	5:	//MoveToTarget ready? -> Druck Ein
		fbMoveToTarget(bExecute:= TRUE);
		IF NOT fbMoveToTarget.bBusy THEN
			IF fbMoveToTarget.bError THEN
				stError.ErrorId := fbMoveToTarget.nErrorId;
				nActionState := 99;
			ELSE
				nActionState := 6;
			END_IF
			fbMoveToTarget(bExecute:= FALSE);
		END_IF	
		
	6:	//Switch Pressure
		IF pStampSupport^.M_GetPressValueOk(nSetPressure:= nPressure1, nTolerancePlus:= 8, nToleranceMinus:= 8) THEN 
			MEMSET(ADR(stActionData),0,SIZEOF(stActionData));
			stActionData.eAction := E_Action.ACTION_SwitchPressure;
			stActionData.aParams[1] := E_PressCtrl.PRESSCTRL_PressOn;
			stError.ErrorId := pStampSupport^.M_ExeAction(stActionData);
		ELSE
			stError.ErrorId := E_ErrorIdCmd.ERRORID_PressTimeOut;
		END_IF
		
		IF stError.ErrorId > 0 THEN	//Error
			stError.ObjectId := pStampSupport^.P_nObjectID;
			nActionState := 99;
		ELSE
			nActionState := 7;
		END_IF

	7:	//MoveZ um ContactDistance nach unten
		nActionState := 8;
		timer1(IN:=FALSE);
		MEMSET(ADR(stActionData),0,SIZEOF(stActionData));
		stActionData.eAction := E_Action.ACTION_MoveZ;
		stActionData.aParams[1] := E_MoveMode.MODE_Relative;
		stActionData.aParams[2] := - nDistance1;
		stActionData.aParams[3] := 1000;
		stError.ErrorId := pStampSupport^.M_ExeAction(stActionData);
		IF stError.ErrorId > 0 THEN	//Error
			stError.ObjectId := pStampSupport^.P_nObjectID;
			nActionState := 99;
		END_IF
		
	8:	//MoveZ ready? -> Timer starten
		IF NOT pStampSupport^.M_GetActionBusy(E_Action.ACTION_MoveZ) THEN
			timer1(IN:=TRUE, PT:= UDINT_TO_TIME(nTime));
			nActionState := 9;
		END_IF
		
	9:	//Warten, bis Zeit abgelaufen -> MoveZ um ContactDistance nach oben
		timer1();
		IF timer1.Q THEN
			nActionState := 10;
			MEMSET(ADR(stActionData),0,SIZEOF(stActionData));
			stActionData.eAction := E_Action.ACTION_MoveZ;
			stActionData.aParams[1] := E_MoveMode.MODE_Relative;
			stActionData.aParams[2] := nDistance1;
			stActionData.aParams[3] := 1000;			
			stError.ErrorId := pStampSupport^.M_ExeAction(stActionData);
			IF stError.ErrorId > 0 THEN	//Error
				stError.ObjectId := pStampSupport^.P_nObjectID;
				nActionState := 99;
			END_IF				
		END_IF
		
	10:	//MoveZ ready? -> Druck aus und MoveFree
		IF NOT pStampSupport^.M_GetActionBusy(E_Action.ACTION_MoveZ) THEN
			MEMSET(ADR(stActionData),0,SIZEOF(stActionData));
			stActionData.eAction := E_Action.ACTION_SwitchPressure;
			stActionData.aParams[1] := 1;
			stActionData.aParams[2] := E_PressCtrl.PRESSCTRL_Off;
			stError.ErrorId := pStampSupport^.M_ExeAction(stActionData);
			IF stError.ErrorId > 0 THEN	//Error
				stError.ObjectId := pStampSupport^.P_nObjectID;
				nActionState := 99;
			ELSE
				stActionData.eAction := E_Action.ACTION_MoveZ;
				stActionData.aParams[1] := E_MoveMode.MODE_Free;
				stActionData.aParams[3] := -1; //MaxSpeed Z
				stError.ErrorId := pStampSupport^.M_ExeAction(stActionData);
				IF stError.ErrorId > 0 THEN	//Error
					stError.ObjectId := pStampSupport^.P_nObjectID;
					nActionState := 99;
				ELSE
					nActionState := 11;
				END_IF			
			END_IF
		END_IF
		
	11:	//MoveZ-Free ready? -> Target = InkStation? -> CloseInkStation
		IF NOT pStampSupport^.M_GetActionBusy(E_Action.ACTION_MoveZ) THEN
			IF pInkStation > 0 THEN
				MEMSET(ADR(stActionData),0,SIZEOF(stActionData));
				stActionData.eAction := E_Action.ACTION_InkOpClCover;
				stActionData.aParams[1] := 1;
				stError.ErrorId := pInkStation^.M_ExeAction(stActionData);
				IF stError.ErrorId > 0 THEN
					stError.ObjectId := pTarget^.P_nObjectID;
					nActionState := 99;
				ELSE
					nActionState := 12;	
				END_IF
			ELSE
				nActionState := 80;
			END_IF
		END_IF
		
	12:	//Inkstation ready? -> Action ready
		IF NOT pInkStation^.M_GetActionBusy(E_Action.ACTION_InkOpClCover) THEN
			nActionState := 80;
		END_IF
		
	70:	//Abbrechen
		nActionState := 80;
		//MoveToTarget oder Einzel-Moves vom MzTool abbrechen (schließen sich gegenseitig aus)
		IF fbMoveToTarget.bBusy THEN
			fbMoveToTarget(bStop:= TRUE);
			nActionState := 70;
		ELSIF pStampSupport^.M_GetActionBusy(E_Action.ACTION_MoveZ) THEN
			pStampSupport^.M_CancelAction(E_Action.ACTION_MoveZ);
			nActionState := 70;
		ELSE
			fbMoveToTarget(bStop:= FALSE);
		END_IF
		
		IF pStampSupport^.M_GetActionBusy(E_Action.ACTION_SetPressure) THEN
			pStampSupport^.M_CancelAction(E_Action.ACTION_SetPressure);
			nActionState := 70;
		END_IF
		
		IF pStampSupport^.M_GetActionBusy(E_Action.ACTION_SwitchPressure) THEN
			pStampSupport^.M_CancelAction(E_Action.ACTION_SwitchPressure);
			nActionState := 70;
		END_IF
		
		//InkStation abbrechen
		IF pInkStation > 0 THEN
			IF pInkStation^.M_GetActionBusy(E_Action.ACTION_InkOpClCover) THEN
				pInkStation^.M_CancelAction(E_Action.ACTION_InkOpClCover);
				nActionState := 70;
			END_IF
		END_IF
END_CASE

//Errorhandling
IF nActionState = 99 THEN
	fbMoveToTarget(bExecute:= FALSE);
	stError.Cmd := E_Action.ACTION_StampInking;
	stError.POUAction := E_POUACT.POUACT_A_StampInking;
	fbErrorList.M_Add(stError);
END_IF
END_ACTION

ACTION A_TeachTarget:
stError.POUState := nActionState;

IF pMzTool^.P_bError THEN
	stError.ErrorId := pMzTool^.P_nErrorId;
	nActionState := 99;
END_IF

IF pMzTool^.P_bCanceled AND nActionState > 0 AND nActionState < 70 THEN
	//MzTool wurde durch StopDevice abgebrochen
	nActionState := 70;
END_IF

CASE nActionState OF
	0:	//MoveToTarget
		IF eTeachOption = E_TeachTrgtOption.Option_PrePos THEN
			MEMSET(ADR(stActionData),0,SIZEOF(stActionData));
			stActionData.eAction := E_Action.ACTION_MoveToTarget;
			stActionData.nObject := pMzTool^.P_nObjectID;
			stActionData.nTarget := pTarget^.P_nObjectID;
		
			IF pTarget^.P_eObjectType = E_ObjectType.OBJECTTYPE_Mtp THEN	//MoveToTarget Well1
				stActionData.aParams[1] := E_TargetRef.TARGETREF_TwoDimArray;
				stActionData.aParams[2] := 1; //Col (erstes Well immer Spalte 1)
				stActionData.aParams[3] := pMtp^.P_nRows; //Row (erstes Well immer letzte Spalte)
			ELSIF pTarget^.P_eObjectType = E_ObjectType.OBJECTTYPE_SpotArray THEN	//MoveToTarget Ecke links unten
				stActionData.aParams[1] := E_TargetRef.TARGETREF_LeftBottom;
			ELSIF pTarget^.P_eObjectType = E_ObjectType.OBJECTTYPE_Slide AND eTargetRef = E_TargetRef.TARGETREF_Alignment THEN	//MoveToTarget Alignment-Marke 1
				stActionData.aParams[1] := E_TargetRef.TARGETREF_SpecPoint;
				stActionData.aParams[2] := 1; //SpecPoint 1 (Marke 1)
			ELSE	//MoveToTarget Slot oder Center
				stActionData.aParams[1] := eTargetRef;
				stActionData.aParams[2] := nSpecPointSlotNr;
			END_IF
			stActionData.aParams[5] := -1;	//MaxSpeed X
			stActionData.aParams[6] := -1;	//MaxSpeed Y
			stActionData.aParams[7] := -1;	//MaxSpeed Z
			stActionData.aParams[10] := nZOffset1;
			stError.ErrorId := fbMoveToTarget.M_SetAndCheckParams(stActionData);
			IF stError.ErrorId > 0 THEN
				nActionState := 99;
			ELSE
				fbMoveToTarget(bExecute:= TRUE);
				nActionState := 1;
			END_IF
			
		ELSIF eTeachOption = E_TeachTrgtOption.Option_NoPrePos THEN
			//alle anderen Tools freifahren
			//dazu wird der Head benötigt:
			stError.ErrorId := pMzTool^.P_pMzHead^.M_MoveFree(pMzTool);
			IF stError.ErrorId > 0 THEN
				nActionState := 99;
			ELSE
				nActionState := 2;
			END_IF
			
		ELSIF eTeachOption = E_TeachTrgtOption.Option_AssumeInstantly THEN
			//aktuellen Wert sofort übernehmen
			stError.ErrorId := pTarget^.M_ApplyPos(eTargetRef, nSpecPointSlotNr, pMzTool^.P_stCurrentPosTotal, bXPos:= TRUE, bYPos:=TRUE, bZPos:=TRUE);
			IF stError.ErrorId > 0 THEN
				nActionState := 99;
			ELSE
				fbObjectDirectory.M_SetObjChange(pTarget^.P_nObjectID);
				nActionState := 80;
			END_IF
		ELSE
			{warnig 'ImplementErrorId'}
			stError.ErrorId := 333;
			nActionState := 99;
		END_IF
		MEMSET(ADR(stInteractRequest),0,SIZEOF(stInteractRequest));

	1:	//MoveToTarget ready?
		fbMoveToTarget(bExecute:= TRUE);
		IF NOT fbMoveToTarget.bBusy THEN
			IF fbMoveToTarget.bError THEN
				stError.ErrorId := fbMoveToTarget.nErrorId;
				nActionState := 99;
			ELSE
				nActionState := 2;	
			END_IF
			fbMoveToTarget(bExecute:= FALSE);
		END_IF
		
	2:	//Interaction Request "StartTeaching"
		IF NOT pMzTool^.P_pMzHead^.M_GetActionBusy(E_Action.ACTION_MoveZ) THEN
			MEMSET(ADR(stInterResponse),0,SIZEOF(stInterResponse));
			stInteractRequest.eInteractMessageType := E_InteractMessageType.INTERACTMES_StartTeaching;
			stInteractRequest.nObjectId := pMzTool^.P_nObjectID;
			stInteractRequest.nArg1 := 1;
			nActionState := 3;
		END_IF
		
	3:	//Response ?
		IF stInterResponse.eInteractMessageType = E_InteractMessageType.INTERACTMES_Assume THEN
			stInteractRequest.nArg1 := stInterResponse.nArg1;
			stInteractRequest.nArg2 := stInterResponse.nArg2;
			stInteractRequest.nArg3 := stInterResponse.nArg3; 
			
			pTarget^.M_ApplyPos(eTargetRef, nSpecPointSlotNr, pMzTool^.P_stCurrentPosTotal,
								bXPos:= DINT_TO_BOOL(stInterResponse.nArg1),
								bYPos:= DINT_TO_BOOL(stInterResponse.nArg2),
								bZPos:= DINT_TO_BOOL(stInterResponse.nArg3));

			fbObjectDirectory.M_SetObjChange(pTarget^.P_nObjectID);
			stInteractRequest.eInteractMessageType := E_InteractMessageType.INTERACTMES_Continue; //Request "Continue"
			MEMSET(ADR(stInterResponse),0,SIZEOF(stInterResponse));

		ELSIF stInterResponse.eInteractMessageType = E_InteractMessageType.INTERACTMES_TeachingFinished THEN
			IF pTarget^.P_eObjectType = E_ObjectType.OBJECTTYPE_Mtp AND eTargetRef = E_TargetRef.TARGETREF_TwoDimArray THEN
				pMtp^.M_CalcOffsetWellLB(pMzTool^.P_stCurrentPosTotal,0);
				stInteractRequest.eInteractMessageType := E_InteractMessageType.INTERACTMES_StartTeaching;	//Request "StartTeaching"
				stInteractRequest.nObjectId := pMzTool^.P_nObjectID;
				stInteractRequest.nArg1 := 2;
				nActionState := 4;
			ELSIF pTarget^.P_eObjectType = E_ObjectType.OBJECTTYPE_SpotArray AND eTargetRef = E_TargetRef.TARGETREF_TwoDimArray THEN
				//Position übertragen (nur XY)
				pTarget^.M_ApplyPos(eTargetRef:= E_TargetRef.TARGETREF_LeftBottom, 0, pMzTool^.P_stCurrentPosTotal,
									bXPos:= TRUE, bYPos:= TRUE, bZPos:= FALSE);
				IF eTeachOption = E_TeachTrgtOption.Option_NoPrePos THEN
					MEMSET(ADR(stInterResponse),0,SIZEOF(stInterResponse));
					stInteractRequest.eInteractMessageType := E_InteractMessageType.INTERACTMES_StartTeaching;	//Request "StartTeaching"
					stInteractRequest.nObjectId := pMzTool^.P_nObjectID;
					stInteractRequest.nArg1 := 2;
					nActionState := 9;
				ELSE
					nActionState := 7; //weiter zu MoveToTarget rechte obere Ecke
				END_IF
			(*
			ELSIF pTarget^.P_eObjectType = E_ObjectType.OBJECTTYPE_Slide AND eTargetRef = E_TargetRef.TARGETREF_Alignment THEN
				//Position auf Marke 1 übertragen
				pSlide := pTarget;
				pSlide^.M_SetMark1Act(pMzTool^.P_stCurrentPosTotal);
				nActionState := 10; //weiter zu MoveToTarget Alignment-Marke 2*)
			ELSE
				nActionState := 20; //weiter zu State "MoveZ-Free"
			END_IF
			MEMSET(ADR(stInterResponse),0,SIZEOF(stInterResponse));
		ELSIF stInterResponse.eInteractMessageType = E_InteractMessageType.INTERACTMES_Cancel THEN
			nActionState := 70;			
		END_IF
		
	//##################################################################################################################
	//Die nächsten 3 Schritte beziehen sich nur auf Mtp mit TargetRef "TwoDimArray"
	//##################################################################################################################
	4:	//Response "TeachingFinished"?
		IF stInterResponse.eInteractMessageType = E_InteractMessageType.INTERACTMES_TeachingFinished THEN
			MEMSET(ADR(stInteractRequest),0,SIZEOF(stInteractRequest));
			//Offset ermitteln und auf Well1 übertragen
			pMtp := pTarget;
			pMtp^.M_CalcOffsetWellLB(pMzTool^.P_stCurrentPosTotal,1);
			//MoveTo Target Wellx
			IF eTeachOption = E_TeachTrgtOption.Option_PrePos THEN
				MEMSET(ADR(stActionData),0,SIZEOF(stActionData));
				stActionData.eAction := E_Action.ACTION_MoveToTarget;
				stActionData.nObject := pMzTool^.P_nObjectID;
				stActionData.nTarget := pMtp^.P_nObjectID;
				stActionData.aParams[1] := E_TargetRef.TARGETREF_TwoDimArray;
				stActionData.aParams[2] := pMtp^.P_nCols; //Col (diagonales Well ermitteln)
				stActionData.aParams[3] := 1; //Row
				stActionData.aParams[5] := -1;	//MaxSpeed X
				stActionData.aParams[6] := -1;	//MaxSpeed Y
				stActionData.aParams[7] := -1;	//MaxSpeed Z
				stError.ErrorId := fbMoveToTarget.M_SetAndCheckParams(stActionData);
				IF stError.ErrorId > 0 THEN
					nActionState := 99;
				ELSE
					fbMoveToTarget(bExecute:= TRUE);
					nActionState := 5;
				END_IF
			ELSE
				MEMSET(ADR(stInterResponse),0,SIZEOF(stInterResponse));
				stInteractRequest.eInteractMessageType := E_InteractMessageType.INTERACTMES_StartTeaching;	//Request "StartTeaching"
				stInteractRequest.nObjectId := pMzTool^.P_nObjectID;
				stInteractRequest.nArg1 := 3;
				nActionState := 6;
			END_IF
		ELSIF stInterResponse.eInteractMessageType = E_InteractMessageType.INTERACTMES_Cancel THEN
			nActionState := 70;
		END_IF
		
	5:	//MoveToTarget ready?
		fbMoveToTarget(bExecute:= TRUE);
		IF NOT fbMoveToTarget.bBusy THEN
			IF fbMoveToTarget.bError THEN
				stError.ErrorId := fbMoveToTarget.nErrorId;
				nActionState := 99;
			ELSE
				MEMSET(ADR(stInterResponse),0,SIZEOF(stInterResponse));
				stInteractRequest.eInteractMessageType := E_InteractMessageType.INTERACTMES_StartTeaching;	//Request "StartTeaching"
				stInteractRequest.nObjectId := pMzTool^.P_nObjectID;
				stInteractRequest.nArg1 := 3;
				nActionState := 6;
			END_IF
			fbMoveToTarget(bExecute:= FALSE);
		END_IF	
		
	6:	//Response "TeachingFinished"?
		IF stInterResponse.eInteractMessageType = E_InteractMessageType.INTERACTMES_TeachingFinished THEN
			//Offset ermitteln und auf Wellx übertragen bzw. Korrekturfaktoren ermitteln
			pMtp^.M_CalcKorrFactor(pMzTool^.P_stCurrentPosTotal);
			nActionState := 20;
		ELSIF stInterResponse.eInteractMessageType = E_InteractMessageType.INTERACTMES_Cancel THEN
			nActionState := 70;
		END_IF
		//##################################################################################################################
		//Ende Teach Mtp Targetref "TwoDimArray
		//##################################################################################################################
		
		//##################################################################################################################
		//Die nächsten 3 Schritte beziehen sich nur auf SpotArray mit TargetRef "TwoDimArray"
		//##################################################################################################################
	7:	//MoveToTarget rechte obere Ecke
		MEMSET(ADR(stActionData),0,SIZEOF(stActionData));
		stActionData.eAction := E_Action.ACTION_MoveToTarget;
		stActionData.nObject := pMzTool^.P_nObjectID;
		stActionData.nTarget := pTarget^.P_nObjectID;
		stActionData.aParams[1] := E_TargetRef.TARGETREF_RightTop;
		stActionData.aParams[5] := -1;	//MaxSpeed X
		stActionData.aParams[6] := -1;	//MaxSpeed Y
		stActionData.aParams[7] := -1;	//MaxSpeed Z
		stActionData.aParams[10] := nZOffset1;
		stError.ErrorId := fbMoveToTarget.M_SetAndCheckParams(stActionData);
		IF stError.ErrorId > 0 THEN
			nActionState := 99;
		ELSE
			fbMoveToTarget(bExecute:= TRUE);
			nActionState := 8;
		END_IF
		
	8:	//MoveToTarget ready?
		fbMoveToTarget(bExecute:= TRUE);
		IF NOT fbMoveToTarget.bBusy THEN
			IF fbMoveToTarget.bError THEN
				stError.ErrorId := fbMoveToTarget.nErrorId;
				nActionState := 99;
			ELSE
				MEMSET(ADR(stInterResponse),0,SIZEOF(stInterResponse));
				stInteractRequest.eInteractMessageType := E_InteractMessageType.INTERACTMES_StartTeaching;	//Request "StartTeaching"
				stInteractRequest.nObjectId := pMzTool^.P_nObjectID;
				stInteractRequest.nArg1 := 2;
				nActionState := 9;
			END_IF
			fbMoveToTarget(bExecute:= FALSE);
		END_IF
		
	9:	//Response "TeachingFinished"?
		IF stInterResponse.eInteractMessageType = E_InteractMessageType.INTERACTMES_TeachingFinished THEN
			//Dimension in XY neu setzen
			stPoint1 := pTarget^.P_stAbsPosLB;
			stPoint2 := pMzTool^.P_stCurrentPosTotal;
			stDimension := pTarget^.P_stDimension;
			stDimension.Width := stPoint2.X - stPoint1.X;
			stDimension.Depth := stPoint2.Y - stPoint1.Y;
			pTarget^.P_stDimension := stDimension;
			nActionState := 20;
		ELSIF stInterResponse.eInteractMessageType = E_InteractMessageType.INTERACTMES_Cancel THEN
			nActionState := 70;
		END_IF	
		//##################################################################################################################
		//Ende Teach SpotArray Targetref "TwoDimArray
		//##################################################################################################################
		

		//##################################################################################################################
		//Die nächsten Schritte beziehen sich nur auf Slide mit TargetRef "Alignment"
		//##################################################################################################################
	10:	//MoveToTarget auf Alignment-Marke 2 Alignment gibt es nicht mehr
		(*
		MEMSET(ADR(stActionData),0,SIZEOF(stActionData));
		stActionData.eAction := E_Action.ACTION_MoveToTarget;
		stActionData.nObject := pMzTool^.P_nObjectID;
		stActionData.nTarget := pTarget^.P_nObjectID;
		stActionData.aParams[1] := E_TargetRef.TARGETREF_SpecPoint;
		stActionData.aParams[2] := 2;	//SpecPoint 1
		stActionData.aParams[5] := -1;	//MaxSpeed X
		stActionData.aParams[6] := -1;	//MaxSpeed Y
		stActionData.aParams[7] := -1;	//MaxSpeed Z
		stActionData.aParams[10] := nZOffset1;
		stError.ErrorId := fbMoveToTarget.M_SetAndCheckParams(stActionData);
		IF stError.ErrorId > 0 THEN
			nActionState := 99;
		ELSE
			fbMoveToTarget(bExecute:= TRUE);
			nActionState := 11;
		END_IF
	
	11:	//MoveToTarget ready?
		fbMoveToTarget(bExecute:= TRUE);
		IF NOT fbMoveToTarget.bBusy THEN
			IF fbMoveToTarget.bError THEN
				stError.ErrorId := fbMoveToTarget.nErrorId;
				nActionState := 99;
			ELSE
				MEMSET(ADR(stInterResponse),0,SIZEOF(stInterResponse));
				stInteractRequest.eInteractMessageType := E_InteractMessageType.INTERACTMES_StartTeaching;	//Request "StartTeaching"
				stInteractRequest.nObjectId := pMzTool^.P_nObjectID;
				stInteractRequest.nArg1 := 2;
				nActionState := 12;
			END_IF
			fbMoveToTarget(bExecute:= FALSE);
		END_IF 
	
	12:	//Response "TeachingFinished"?
		IF stInterResponse.eInteractMessageType = E_InteractMessageType.INTERACTMES_TeachingFinished THEN
			pSlide^.M_SetMark2Act(pMzTool^.P_stCurrentPosTotal);
			//Winkel berechnen
			pSlide^.P_bIsAligned := TRUE;
			pSlide^.M_CalcAngle();
			nActionState := 20;
		ELSIF stInterResponse.eInteractMessageType = E_InteractMessageType.INTERACTMES_Cancel THEN
			pSlide^.P_bIsAligned := FALSE;
			nActionState := 70;
		END_IF*)

	20:	//MoveZ-Free
		//Falls das Tool am unteren Head ist, dann freifahren überspringen.
		nActionState := 21;
		IF pMzTool^.P_pMzHead^.P_bIsTopHead THEN
			MEMSET(ADR(stActionData),0,SIZEOF(stActionData));
			stActionData.eAction := E_Action.ACTION_MoveZ;
			stActionData.aParams[1] := E_MoveMode.MODE_Free;
			stActionData.aParams[3] := -1;	//MaxSpeed Z
			stError.ErrorId := pMzTool^.M_ExeAction(stActionData);
			IF stError.ErrorId > 0 THEN
				nActionState := 99;
			END_IF
		END_IF
	
	21:	//MoveZ-Free ready? -> Action ready
		IF NOT pMzTool^.M_GetActionBusy(E_Action.ACTION_MoveZ) THEN
			fbObjectDirectory.M_SetObjChange(pTarget^.P_nObjectID);
			nActionState := 80;
			MEMSET(ADR(stInteractRequest),0,SIZEOF(stInteractRequest));
		END_IF
	
	70:	//Abbrechen
		IF fbMoveToTarget.bBusy THEN
			fbMoveToTarget(bStop:= TRUE);
		ELSIF pMzTool^.M_GetActionBusy(E_Action.ACTION_MoveZ) THEN
			pMzTool^.M_CancelAction(E_Action.ACTION_MoveZ);
		ELSE
			fbMoveToTarget(bExecute:= FALSE);
			MEMSET(ADR(stInteractRequest),0,SIZEOF(stInteractRequest));
			nActionState := 80;
		END_IF
END_CASE

//Errorhandling
IF nActionState = 99 THEN
	fbMoveToTarget(bExecute:= FALSE);
	stError.ObjectId := pMzTool^.P_nObjectID;
	stError.Cmd := E_Action.ACTION_TeachTarget;
	stError.POUAction := E_POUACT.POUACT_A_TeachTarget;
	fbErrorList.M_Add(stError);
END_IF
END_ACTION

ACTION A_TeachTool:
stError.POUState := nActionState;

IF pMzTool^.P_bError THEN
	stError.ErrorId := pMzTool^.P_nErrorId;
	nActionState := 99;
END_IF

IF pMzTool^.P_bCanceled AND nActionState > 0 AND nActionState < 70 THEN
	//MzTool wurde durch StopDevice abgebrochen
	nActionState := 70;
END_IF

CASE nActionState OF
	0:	//MoveToTarget
		MEMSET(ADR(stActionData),0,SIZEOF(stActionData));
		//stActionData.bIntern := TRUE;
		stActionData.eAction := E_Action.ACTION_MoveToTarget;
		stActionData.nObject := pMzTool^.P_nObjectID;
		stActionData.nTarget := pTarget^.P_nObjectID;
    	stActionData.aParams[1] := eTargetRef;
		stActionData.aParams[2] := nCol;
		stActionData.aParams[3] := nRow;
		stActionData.aParams[5] := -1;	//MaxSpeed X
		stActionData.aParams[6] := -1;	//MaxSpeed Y
		stActionData.aParams[7] := -1;	//MaxSpeed Z
		stActionData.aParams[10] := nZOffset1;		

		stError.ErrorId := fbMoveToTarget.M_SetAndCheckParams(stActionData);
		IF stError.ErrorId > 0 THEN
			nActionState := 99;
		ELSE
			fbMoveToTarget(bExecute:= TRUE);
			MEMSET(ADR(stInteractRequest),0,SIZEOF(stInteractRequest));
			nActionState := 1;
		END_IF		

	1:	//MoveToTarget ready? -> Request "StartTeaching"
		fbMoveToTarget(bExecute:= TRUE);
		IF NOT fbMoveToTarget.bBusy THEN
			IF fbMoveToTarget.bError THEN
				stError.ErrorId := fbMoveToTarget.nErrorId;
				nActionState := 99;
			ELSE
				MEMSET(ADR(stInterResponse),0,SIZEOF(stInterResponse));
				stInteractRequest.eInteractMessageType := E_InteractMessageType.INTERACTMES_StartTeaching;	//Interaction Request absenden
				stInteractRequest.nObjectId := pMzTool^.P_nObjectID;
				stInteractRequest.nArg1 := 1;
				nActionState := 2;
			END_IF
			fbMoveToTarget(bExecute:= FALSE);
		END_IF
	
	2:	//Zwischenschritt um stInteractRequest zurückzusetzen
		MEMSET(ADR(stInteractRequest),0,SIZEOF(stInteractRequest));
		nActionState := 3;

	3:	//Response ?
		IF stInterResponse.eInteractMessageType = E_InteractMessageType.INTERACTMES_Assume THEN
			//anhand von den Args von Response wird festgelegt, ob die Werte von X,Y,Z übernommen werden sollen
			//absolute Position (Sollposition)aus Target holen
			stPoint1 := pTarget^.M_GetAbsPos(pChildPos:= 0, eTargetRef:= eTargetRef,
												nParam1:= nCol, nParam2:= nRow, nParam3:= 0,nZLevel:= 0);			
			IF stInterResponse.nArg1 = 1 THEN
				pMzTool^.M_SetCurrentPos(1,stPoint1.X);
				stInteractRequest.nArg1 := 1;			
			END_IF

			IF stInterResponse.nArg2 = 1 THEN
				pMzTool^.M_SetCurrentPos(2,stPoint1.Y);
				stInteractRequest.nArg2 := 1;
			END_IF

			IF stInterResponse.nArg3 = 1 THEN
				pMzTool^.M_SetCurrentPos(3,stPoint1.Z);
				stInteractRequest.nArg3 := 1;
			END_IF
			stInteractRequest.eInteractMessageType := E_InteractMessageType.INTERACTMES_Continue;	//Request "Continue"
			MEMSET(ADR(stInterResponse),0,SIZEOF(stInterResponse));
		ELSIF stInterResponse.eInteractMessageType = E_InteractMessageType.INTERACTMES_TeachingFinished OR 
				stInterResponse.eInteractMessageType = E_InteractMessageType.INTERACTMES_Cancel THEN
			MEMSET(ADR(stInteractRequest),0,SIZEOF(stInteractRequest));
			MEMSET(ADR(stInterResponse),0,SIZEOF(stInterResponse));				
			nActionState := 80;
		END_IF

	70:	//Abbrechen
		IF fbMoveToTarget.bBusy THEN
			fbMoveToTarget(bStop:= TRUE);
		ELSE
			fbMoveToTarget(bExecute:= FALSE);
			MEMSET(ADR(stInteractRequest),0,SIZEOF(stInteractRequest));
			MEMSET(ADR(stInterResponse),0,SIZEOF(stInterResponse));
			nActionState := 80;
		END_IF		
END_CASE

//Errorhandling
IF nActionState = 99 THEN
	fbMoveToTarget(bExecute:= FALSE);
	stError.ObjectId := pMzTool^.P_nObjectID;
	stError.Cmd := E_Action.ACTION_TeachTool;
	stError.POUAction := E_POUACT.POUACT_A_TeachTool;
	fbErrorList.M_Add(stError);
END_IF
END_ACTION

ACTION A_TransferGas:
stError.POUState := nActionState;

IF pLuer^.P_bError THEN
	stError.ObjectId := pLuer^.P_nObjectID;
	stError.ErrorId := pLuer^.P_nErrorId;
	nActionState := 99;
ELSIF pLuer2^.P_bError THEN
	stError.ObjectId := pLuer2^.P_nObjectID;
	stError.ErrorId := pLuer2^.P_nErrorId;
	nActionState := 99;	
END_IF

IF (pLuer^.P_bCanceled OR pLuer2^.P_bCanceled) AND nActionState > 0 AND nActionState < 70 THEN
	//Ein MzTool wurde durch StopDevice abgebrochen
	nActionState := 70;
END_IF

CASE nActionState OF
	0:	//Voreinstellung Ventile

		//LuerSource
		//ValveDil on
		pLuer^.M_SwitchValveDiluter(TRUE);
		
		//ValveLuer off
		pLuer^.M_SwitchValveLuer(FALSE);
		
		//LuerDestination
		//ValveDil off
		pLuer2^.M_SwitchValveDiluter(FALSE);
		
		//ValveLuer on
		pLuer2^.M_SwitchValveLuer(TRUE);
		
		//Druck einstellen
		MEMSET(ADR(stActionData),0,SIZEOF(stActionData));
		stActionData.eAction := E_Action.ACTION_SetPressure;
		stActionData.aParams[1] := 1; //Fertigmeldung wenn Solldruck erreicht
		stActionData.aParams[2] := nPressure1; //Value in kPa
		stActionData.aParams[3] := 15; //Toleranz
		stActionData.aParams[4] := 15; //Toleranz
		stActionData.aParams[5] := 10000; //Timeout in ms
		stError.ErrorId :=  pLuer^.M_ExeAction(stActionData);
		IF stError.ErrorId > 0 THEN
			stError.ObjectId := pLuer^.P_nObjectID;
			nActionState := 99;
		ELSE
			nActionState := 1;
		END_IF
	
	1:	//Start Timer, ValveSynth.Gas "On"
		IF NOT pLuer^.M_GetActionBusy(E_Action.ACTION_SetPressure) THEN
			timer1(IN:=TRUE,PT:= DWORD_TO_TIME(nTime));
			pLuer^.M_SwitchValveSynthGas(TRUE);
			nActionState := 2;
		END_IF
		
	2:	//Timer ready? -> ValveSynth.Gas "Off"
		timer1();
		IF timer1.Q THEN
			timer1(IN:=FALSE);
			pLuer^.M_SwitchValveSynthGas(FALSE);
			pLuer^.M_SwitchValveDiluter(FALSE);
			pLuer2^.M_SwitchValveLuer(FALSE);
			nActionState := 80;
		END_IF
		
	70:	//Abbrechen
		nActionState := 80;
		IF pLuer^.M_GetActionBusy(E_Action.ACTION_SetPressure) THEN
			pLuer^.M_CancelAction(E_Action.ACTION_SetPressure);
			nActionState := 70;
		END_IF
		timer1(IN:=FALSE);
		pLuer^.M_SwitchValveSynthGas(FALSE);
		pLuer^.M_SwitchValveDiluter(FALSE);
		pLuer2^.M_SwitchValveLuer(FALSE);
END_CASE

//Errorhandling
IF nActionState = 99 THEN
	stError.Cmd := E_Action.ACTION_TransferGas;
	stError.POUAction := E_POUACT.POUACT_A_TransferGas;
	fbErrorList.M_Add(stError);
END_IF
END_ACTION

ACTION A_TransferLiquid:
stError.POUState := nActionState;

IF pDiluter1^.P_bError THEN
	stError.ErrorId := pDiluter1^.P_nErrorId;
	nActionState := 99;
END_IF

IF (pDiluter1^.P_bCanceled OR pLuer^.P_bCanceled OR pLuer2^.P_bCanceled) AND nActionState > 0 AND nActionState < 70 THEN
	//Ein MzTool wurde durch StopDevice abgebrochen
	nActionState := 70;
END_IF

CASE nActionState OF
	0:	//Voreinstellung Ventile
		//LuerSource
		//ValveDil on
		pLuer^.M_SwitchValveDiluter(TRUE);
		//ValveLuer on
		pLuer^.M_SwitchValveLuer(TRUE);
		//LuerDestination
		//ValveDil off
		pLuer2^.M_SwitchValveDiluter(TRUE);
		//ValveLuer on
		pLuer2^.M_SwitchValveLuer(TRUE);
		
		//Transfer am DilSource ausführen
		MEMSET(ADR(stActionData),0,SIZEOF(stActionData));
		stActionData.eAction := E_Action.ACTION_DilTransfer;
		stActionData.aParams[1] := pDiluter2^.P_nObjectID; //ObjectId DilDesti
		stActionData.aParams[2] := nQuantity1;
		stActionData.aParams[3] := nFlow1;
		stActionData.aParams[4] := nQuantity2;
		stActionData.aParams[5] := nQuantity3;

		stError.ErrorId :=  pDiluter1^.M_ExeAction(stActionData);
		IF stError.ErrorId > 0 THEN
			stError.ObjectId := pDiluter1^.P_nObjectID;
			nActionState := 99;
		ELSE
			nActionState := 1;
		END_IF		
		
	1:	//Transfer ready?
		IF NOT pDiluter1^.M_GetActionBusy(E_Action.ACTION_DilTransfer) THEN
			pLuer^.M_SwitchValveDiluter(FALSE);
			pLuer^.M_SwitchValveLuer(FALSE);
			pLuer2^.M_SwitchValveDiluter(FALSE);
			pLuer2^.M_SwitchValveLuer(FALSE);
			nActionState := 80;
		END_IF
	
	70:	//Abbrechen
		IF pDiluter1^.M_GetActionBusy(E_Action.ACTION_DilTransfer) THEN
			pDiluter1^.M_CancelAction(E_Action.ACTION_DilTransfer);
		ELSE
			pLuer^.M_SwitchValveDiluter(FALSE);
			pLuer^.M_SwitchValveLuer(FALSE);
			pLuer2^.M_SwitchValveDiluter(FALSE);
			pLuer2^.M_SwitchValveLuer(FALSE);
			nActionState := 80;			
		END_IF
END_CASE

//Errorhandling
IF nActionState = 99 THEN
	stError.Cmd := E_Action.ACTION_TransferLiquid;
	stError.POUAction := E_POUACT.POUACT_A_TransferLiquid;
	fbErrorList.M_Add(stError);
END_IF
END_ACTION

ACTION A_TransferTray:
//Mögliche Transfers
//-von linker Übergabestation zu TrayTransporterSlot
//-von rechter Übergabestation zu TrayTransporterSlot
//-von TrayTransporterSlot zu linker Übergabestation
//-von TrayTransporterSlot zu rechter Übergabestation

//Der Error muss für die States 0-2 hier gemeldet werden
//sonst erfolgt die Meldung aus den Sub-Actions
IF nActionState < 3 THEN
	IF pTrayTransporter^.P_bError THEN
		stError.ErrorId := pTrayTransporter^.P_nErrorId;
		stError.ObjectId := pTrayTransporter^.P_nObjectID;
		stError.Cmd := E_Action.ACTION_TransferTray;
		stError.POUAction := E_POUACT.POUACT_A_TransferTray;
		fbErrorList.M_Add(stError);
		nActionState := 99;	
	END_IF	
END_IF

IF nActionState > 0 AND nActionState < 70 AND pTrayTransporter^.P_bCanceled THEN
	nActionState := 70;
END_IF

CASE nActionState OF
	0:	//Both DrivingPins horizontal
		MEMSET(ADR(stActionData),0,SIZEOF(stActionData));
		stActionData.eAction := E_Action.ACTION_TurnDrivingPin;
		stActionData.nObject := pTrayTransporter^.P_nObjectID;
		stActionData.aParams[1] := E_DrivingPinSelection.Both;
		stActionData.aParams[2] := E_DrivingPinCtrl.Horizontal;
		stError.ErrorId := pTrayTransporter^.M_ExeAction(stActionData);
		IF stError.ErrorId > 0 THEN
			nActionState := 99;
		ELSE
			nActionState := 1;
		END_IF
		
	1:	//DrivingPins ready? -> Unlock TrayLock
		IF NOT pTrayTransporter^.M_GetActionBusy(E_Action.ACTION_TurnDrivingPin) THEN
			MEMSET(ADR(stActionData),0,SIZEOF(stActionData));
			stActionData.eAction := E_Action.ACTION_LockUnlock;
			stActionData.aParams[1] := E_LockCtrl.Unlock;
			stError.ErrorId := pTrayTransporter^.M_ExeAction(stActionData);
			IF stError.ErrorId > 0 THEN
				nActionState := 99;
			ELSE
				nActionState := 2;
			END_IF
		END_IF
		
	2:	//TrayLock ready?
		IF NOT pTrayTransporter^.M_GetActionBusy(E_Action.ACTION_LockUnlock) THEN
			IF pTrayTransporter^.P_bError THEN
				nActionState := 99;
			ELSE
				CASE eTransferTrayCtrl OF
					E_TransferTrayCtrl.LeftToSlot:
						nActionState := 3;
					E_TransferTrayCtrl.RightToSlot:
						nActionState := 4;
					E_TransferTrayCtrl.SlotToLeft:
						nActionState := 5;
					E_TransferTrayCtrl.SlotToRight:
						nActionState := 6;
				END_CASE
			END_IF
		END_IF
		
	3:	//Transfer left to slot
		A_TransferTrayLeftToSlot();
		IF nStateA_TransferTray >= 80 THEN
			IF nStateA_TransferTray = 99 THEN
				nActionState := 99;
			ELSE
				nActionState := 80;
			END_IF
			nStateA_TransferTray := 0;
		END_IF
	
	4:	//Transfer right to slot
		A_TransferTrayRightToSlot();
		IF nStateA_TransferTray >= 80 THEN
			IF nStateA_TransferTray = 99 THEN
				nActionState := 99;
			ELSE
				nActionState := 80;
			END_IF
			nStateA_TransferTray := 0;
		END_IF
	
	5:	//Transfer slot to left
		A_TransferTraySlotToLeft();
		IF nStateA_TransferTray >= 80 THEN
			IF nStateA_TransferTray = 99 THEN
				nActionState := 99;
			ELSE
				nActionState := 80;
			END_IF
			nStateA_TransferTray := 0;
		END_IF
	
	6:	//Transfer slot to right
		A_TransferTraySlotToRight();
		IF nStateA_TransferTray >= 80 THEN
			IF nStateA_TransferTray = 99 THEN
				nActionState := 99;
			ELSE
				nActionState := 80;
			END_IF
			nStateA_TransferTray := 0;
		END_IF
		
	70:	//Abbrechen
		IF pTrayTransporter^.P_bBusy THEN
			pTrayTransporter^.M_Stop();
		ELSE
			nStateA_TransferTray := 0;
			nActionState := 80;
		END_IF
END_CASE
END_ACTION

ACTION A_TransferTrayLeftToSlot:
CASE nStateA_TransferTray OF
	0:	//TransferStation ready for transfer?
		stError.ErrorId := pTrayTransporter^.M_GetStateForTransfer(E_TransferTrayCtrl.LeftToSlot);
		IF stError.ErrorId = 0 THEN
			nStateA_TransferTray := 1;
		ELSE
			nStateA_TransferTray := 99;
		END_IF
		
	1:	//Move slider TransferPosition left
		stActionData.eAction := E_Action.ACTION_MoveTrayTransporter;
		stActionData.aParams[1] := pTrayTransporter^.P_nTransferPosLeft;
		stActionData.aParams[2] := pTrayTransporter^.P_nMaxSliderSpeed;
		stError.ErrorId := pTrayTransporter^.M_ExeAction(stActionData);
		IF stError.ErrorId > 0 THEN
			nStateA_TransferTray := 99;
		ELSE
			nStateA_TransferTray := 2;
		END_IF
		
	2:	//Move ready? DrivingPin left vertical
		IF NOT pTrayTransporter^.M_GetActionBusy(E_Action.ACTION_MoveTrayTransporter) THEN
			stActionData.eAction := E_Action.ACTION_TurnDrivingPin;
			stActionData.aParams[1] := E_DrivingPinSelection.Left;
			stActionData.aParams[2] := E_DrivingPinCtrl.Vertical;
			stError.ErrorId := pTrayTransporter^.M_ExeAction(stActionData);
			IF stError.ErrorId > 0 THEN
				nStateA_TransferTray := 99;
			ELSE
				nStateA_TransferTray := 3;
			END_IF
		END_IF
		
	3:	//TurnDrivingPin ready? -> Move slider to slot + gap
		//Hier kann es sein, dass es nicht mit einem Zug geht.
		//Wenn also die TransferPos > als max SliderPos ist, dann wird zuerst bis max. Pos gefahren und dann über die mittlere Aussparung
		//das benötigt zusätzliche Steps
		IF NOT pTrayTransporter^.M_GetActionBusy(E_Action.ACTION_TurnDrivingPin) THEN
			stActionData.eAction := E_Action.ACTION_MoveTrayTransporter;
			nTransferTrayPos := pTrayTransporter^.M_GetSliderPosTrayInSlot(E_DrivingPinSelection.Left, E_TrayHollowSelection.Right) + pTrayTransporter^.P_nDrivingPinGap;
			IF nTransferTrayPos > pTrayTransporter^.P_nMaxSliderPos THEN
				nTransferTrayPos := pTrayTransporter^.P_nMaxSliderPos;
				nStateA_TransferTray := 4;
			ELSE
				nStateA_TransferTray := 20;
			END_IF
			stActionData.aParams[1] := nTransferTrayPos;
			stActionData.aParams[2] := cMoveTraySpeed;
			stError.ErrorId := pTrayTransporter^.M_ExeAction(stActionData);
			IF stError.ErrorId > 0 THEN
				nStateA_TransferTray := 99;
			END_IF
		END_IF
		
	4:	//Move ready? -> Move slider centre hollow (last pos - gap)
		IF NOT pTrayTransporter^.M_GetActionBusy(E_Action.ACTION_MoveTrayTransporter) THEN
			stActionData.eAction := E_Action.ACTION_MoveTrayTransporter;
			nTransferTrayPos :=  nTransferTrayPos - pTrayTransporter^.P_nDrivingPinGap;
			stActionData.aParams[1] := nTransferTrayPos;
			stActionData.aParams[2] := pTrayTransporter^.P_nMaxSliderSpeed;
			stError.ErrorId := pTrayTransporter^.M_ExeAction(stActionData);
			IF stError.ErrorId > 0 THEN
				nStateA_TransferTray := 99;
			ELSE
				nStateA_TransferTray := 5;
			END_IF
		END_IF
		
	5:	//Move ready? DrivingPinLeft horizontal
		IF NOT pTrayTransporter^.M_GetActionBusy(E_Action.ACTION_MoveTrayTransporter) THEN
			stActionData.eAction := E_Action.ACTION_TurnDrivingPin;
			stActionData.aParams[1] := E_DrivingPinSelection.Left;
			stActionData.aParams[2] := E_DrivingPinCtrl.Horizontal;
			stError.ErrorId := pTrayTransporter^.M_ExeAction(stActionData);
			IF stError.ErrorId > 0 THEN
				nStateA_TransferTray := 99;
			ELSE
				nStateA_TransferTray := 6;
			END_IF
		END_IF
		
	6:	//TurnDrivingPin ready? -> Move slider centre of tray (relative)
		IF NOT pTrayTransporter^.M_GetActionBusy(E_Action.ACTION_TurnDrivingPin) THEN
			stActionData.eAction := E_Action.ACTION_MoveTrayTransporter;
			nTransferTrayPos := nTransferTrayPos - pTrayTransporter^.P_nTrayLength /2 + pTrayTransporter^.P_nHollowDistance;
			stActionData.aParams[1] := nTransferTrayPos;
			stActionData.aParams[2] := pTrayTransporter^.P_nMaxSliderSpeed;
			stError.ErrorId := pTrayTransporter^.M_ExeAction(stActionData);
			IF stError.ErrorId > 0 THEN
				nStateA_TransferTray := 99;
			ELSE
				nStateA_TransferTray := 7;
			END_IF
		END_IF
		
	7:	//Move ready? DrivingPinLeft vertical
		IF NOT pTrayTransporter^.M_GetActionBusy(E_Action.ACTION_MoveTrayTransporter) THEN
			stActionData.eAction := E_Action.ACTION_TurnDrivingPin;
			stActionData.aParams[1] := E_DrivingPinSelection.Left;
			stActionData.aParams[2] := E_DrivingPinCtrl.Vertical;
			stError.ErrorId := pTrayTransporter^.M_ExeAction(stActionData);
			IF stError.ErrorId > 0 THEN
				nStateA_TransferTray := 99;
			ELSE
				nStateA_TransferTray := 8;
			END_IF
		END_IF
		
	8:	//TurnDrivingPin ready? -> Move slider to Slot
		IF NOT pTrayTransporter^.M_GetActionBusy(E_Action.ACTION_TurnDrivingPin) THEN
			stActionData.eAction := E_Action.ACTION_MoveTrayTransporter;
			nTransferTrayPos := pTrayTransporter^.M_GetSliderPosTrayInSlot(E_DrivingPinSelection.Left, E_TrayHollowSelection.Centre) + pTrayTransporter^.P_nDrivingPinGap;
			stActionData.aParams[1] := nTransferTrayPos;
			stActionData.aParams[2] := cMoveTraySpeed;
			stError.ErrorId := pTrayTransporter^.M_ExeAction(stActionData);
			IF stError.ErrorId > 0 THEN
				nStateA_TransferTray := 99;
			ELSE
				nStateA_TransferTray := 20;
			END_IF
		END_IF
		
	
	//Hier wird die Abzweigung in State "3" wieder zusammengeführt
		
	20:	//Move ready? -> Move slider centre hollow (last pos - gap)
		IF NOT pTrayTransporter^.M_GetActionBusy(E_Action.ACTION_MoveTrayTransporter) THEN
			stActionData.eAction := E_Action.ACTION_MoveTrayTransporter;
			stActionData.aParams[1] := nTransferTrayPos - pTrayTransporter^.P_nDrivingPinGap;
			stActionData.aParams[2] := pTrayTransporter^.P_nMaxSliderSpeed;
			stError.ErrorId := pTrayTransporter^.M_ExeAction(stActionData);
			IF stError.ErrorId > 0 THEN
				nStateA_TransferTray := 99;
			ELSE
				nStateA_TransferTray := 21;
			END_IF
		END_IF
		
	21:	//Move ready? DrivingPinLeft horizontal
		IF NOT pTrayTransporter^.M_GetActionBusy(E_Action.ACTION_MoveTrayTransporter) THEN
			stActionData.eAction := E_Action.ACTION_TurnDrivingPin;
			stActionData.aParams[1] := E_DrivingPinSelection.Left;
			stActionData.aParams[2] := E_DrivingPinCtrl.Horizontal;
			stError.ErrorId := pTrayTransporter^.M_ExeAction(stActionData);
			IF stError.ErrorId > 0 THEN
				nStateA_TransferTray := 99;
			ELSE
				nStateA_TransferTray := 22;
			END_IF
		END_IF

	22:	//TurnDrivingPin ready? -> Lock TrayLock
		IF NOT pTrayTransporter^.M_GetActionBusy(E_Action.ACTION_TurnDrivingPin) THEN
			stActionData.eAction := E_Action.ACTION_LockUnlock;
			stActionData.aParams[1] := E_LockCtrl.Lock;
			stError.ErrorId := pTrayTransporter^.M_ExeAction(stActionData);
			IF stError.ErrorId > 0 THEN
				nStateA_TransferTray := 99;
			ELSE
				nStateA_TransferTray := 23;
			END_IF
		END_IF
		
	23:	//TrayLock ready? -> Action ready
		IF NOT pTrayTransporter^.M_GetActionBusy(E_Action.ACTION_LockUnlock) THEN
			nStateA_TransferTray := 80;
		END_IF
END_CASE

//Errorhandling
IF nStateA_TransferTray = 99 THEN
	stError.Cmd := E_Action.ACTION_TransferTray;
	stError.POUAction := E_POUACT.POUACT_A_TransferTrayLeftToSlot;
	fbErrorList.M_Add(stError);	
END_IF
END_ACTION

ACTION A_TransferTrayRightToSlot:
CASE nStateA_TransferTray OF
	0:	//TransferStation ready for transfer?
		stError.ErrorId := pTrayTransporter^.M_GetStateForTransfer(E_TransferTrayCtrl.RightToSlot);
		IF stError.ErrorId = 0 THEN
			nStateA_TransferTray := 1;
		ELSE
			nStateA_TransferTray := 99;
		END_IF
		
	1:	//Move slider TransferPosition right
		stActionData.eAction := E_Action.ACTION_MoveTrayTransporter;
		stActionData.aParams[1] := pTrayTransporter^.P_nTransferPosRight;
		stActionData.aParams[2] := pTrayTransporter^.P_nMaxSliderSpeed;
		stError.ErrorId := pTrayTransporter^.M_ExeAction(stActionData);
		IF stError.ErrorId > 0 THEN
			nStateA_TransferTray := 99;
		ELSE
			nStateA_TransferTray := 2;
		END_IF
		
	2:	//Move ready? DrivingPin right vertical
		IF NOT pTrayTransporter^.M_GetActionBusy(E_Action.ACTION_MoveTrayTransporter) THEN
			stActionData.eAction := E_Action.ACTION_TurnDrivingPin;
			stActionData.aParams[1] := E_DrivingPinSelection.Right;
			stActionData.aParams[2] := E_DrivingPinCtrl.Vertical;
			stError.ErrorId := pTrayTransporter^.M_ExeAction(stActionData);
			IF stError.ErrorId > 0 THEN
				nStateA_TransferTray := 99;
			ELSE
				nStateA_TransferTray := 3;
			END_IF
		END_IF
		
	3:	//TurnDrivingPin ready? -> Move slider to SafePosLeft
		//Zuerst soweit wie möglich nach links fahren und dann um Abstand der äußeren Aussparungen wieder nach rechts fahren
		IF NOT pTrayTransporter^.M_GetActionBusy(E_Action.ACTION_TurnDrivingPin) THEN
			stActionData.eAction := E_Action.ACTION_MoveTrayTransporter;
			nTransferTrayPos := pTrayTransporter^.P_nSafePosLeft;
			stActionData.aParams[1] := nTransferTrayPos;
			stActionData.aParams[2] := cMoveTraySpeed;
			stError.ErrorId := pTrayTransporter^.M_ExeAction(stActionData);
			IF stError.ErrorId > 0 THEN
				nStateA_TransferTray := 99;
			ELSE
				nStateA_TransferTray := 4;
			END_IF
		END_IF
		
	4:	//Move ready? -> Move slider centre hollow (last pos + gap)
		IF NOT pTrayTransporter^.M_GetActionBusy(E_Action.ACTION_MoveTrayTransporter) THEN
			stActionData.eAction := E_Action.ACTION_MoveTrayTransporter;
			nTransferTrayPos :=  nTransferTrayPos + pTrayTransporter^.P_nDrivingPinGap;
			stActionData.aParams[1] := nTransferTrayPos;
			stActionData.aParams[2] := pTrayTransporter^.P_nMaxSliderSpeed;
			stError.ErrorId := pTrayTransporter^.M_ExeAction(stActionData);
			IF stError.ErrorId > 0 THEN
				nStateA_TransferTray := 99;
			ELSE
				nStateA_TransferTray := 5;
			END_IF
		END_IF
		
	5:	//Move ready? DrivingPinRight horizontal
		IF NOT pTrayTransporter^.M_GetActionBusy(E_Action.ACTION_MoveTrayTransporter) THEN
			stActionData.eAction := E_Action.ACTION_TurnDrivingPin;
			stActionData.aParams[1] := E_DrivingPinSelection.Right;
			stActionData.aParams[2] := E_DrivingPinCtrl.Horizontal;
			stError.ErrorId := pTrayTransporter^.M_ExeAction(stActionData);
			IF stError.ErrorId > 0 THEN
				nStateA_TransferTray := 99;
			ELSE
				nStateA_TransferTray := 6;
			END_IF
		END_IF
		
	6:	//Right hollow reachable?
		IF NOT pTrayTransporter^.M_GetActionBusy(E_Action.ACTION_TurnDrivingPin) THEN
			IF bAdditionalMoves THEN
				IF nTransferTrayPos + pTrayTransporter^.P_nHollowToHollow / 2 <= pTrayTransporter^.P_nMaxSliderPos THEN
					nStateA_TransferTray := 10;
				ELSE
					stError.ErrorId := E_ErrorIdCmd.ERRORID_CanNotTransferTrayCompletely;
					nStateA_TransferTray := 99; 
				END_IF
			ELSE
				IF nTransferTrayPos + pTrayTransporter^.P_nHollowToHollow <= pTrayTransporter^.P_nMaxSliderPos  THEN
					nStateA_TransferTray := 10;
				ELSE
					nStateA_TransferTray := 7;
				END_IF
			END_IF
		END_IF
		
	7:	//Move slider to middle hollow
		stActionData.eAction := E_Action.ACTION_MoveTrayTransporter;
		nTransferTrayPos := nTransferTrayPos + pTrayTransporter^.P_nTrayLength/2 - pTrayTransporter^.P_nHollowDistance;
		stActionData.aParams[1] := nTransferTrayPos;
		stActionData.aParams[2] := pTrayTransporter^.P_nMaxSliderSpeed;
		stError.ErrorId := pTrayTransporter^.M_ExeAction(stActionData);
		IF stError.ErrorId > 0 THEN
			nStateA_TransferTray := 99;
		ELSE
			nStateA_TransferTray := 8;
		END_IF
		
	8:	//Move ready? DrivingPin right vertical
		IF NOT pTrayTransporter^.M_GetActionBusy(E_Action.ACTION_MoveTrayTransporter) THEN
			stActionData.eAction := E_Action.ACTION_TurnDrivingPin;
			stActionData.aParams[1] := E_DrivingPinSelection.Right;
			stActionData.aParams[2] := E_DrivingPinCtrl.Vertical;
			stError.ErrorId := pTrayTransporter^.M_ExeAction(stActionData);
			IF stError.ErrorId > 0 THEN
				nStateA_TransferTray := 99;
			ELSE
				nStateA_TransferTray := 9;
			END_IF
		END_IF
		
	9:	//TurnDrivingPin ready? -> Move SafePosL
		IF NOT pTrayTransporter^.M_GetActionBusy(E_Action.ACTION_TurnDrivingPin) THEN
			stActionData.eAction := E_Action.ACTION_MoveTrayTransporter;
			nTransferTrayPos := pTrayTransporter^.P_nSafePosLeft;
			stActionData.aParams[1] := nTransferTrayPos;
			stActionData.aParams[2] := cMoveTraySpeed;
			stError.ErrorId := pTrayTransporter^.M_ExeAction(stActionData);
			IF stError.ErrorId > 0 THEN
				nStateA_TransferTray := 99;
			ELSE
				bAdditionalMoves := TRUE;
				nStateA_TransferTray := 4;
			END_IF
		END_IF

	10:	//TurnDrivingPin ready? -> Move slider at distance of both hollows (relative to previous position)
		stActionData.eAction := E_Action.ACTION_MoveTrayTransporter;
		IF bAdditionalMoves THEN //wird in State
			nTransferTrayPos := nTransferTrayPos + pTrayTransporter^.P_nHollowToHollow / 2;
		ELSE
			nTransferTrayPos := nTransferTrayPos + pTrayTransporter^.P_nHollowToHollow;	
		END_IF
		stActionData.aParams[1] := nTransferTrayPos;
		stActionData.aParams[2] := pTrayTransporter^.P_nMaxSliderSpeed;
		stError.ErrorId := pTrayTransporter^.M_ExeAction(stActionData);
		IF stError.ErrorId > 0 THEN
			nStateA_TransferTray := 99;
		ELSE
			nStateA_TransferTray := 11;
		END_IF
		
	11:	//Move ready? DrivingPinRight vertical
		IF NOT pTrayTransporter^.M_GetActionBusy(E_Action.ACTION_MoveTrayTransporter) THEN
			stActionData.eAction := E_Action.ACTION_TurnDrivingPin;
			stActionData.aParams[1] := E_DrivingPinSelection.Right;
			stActionData.aParams[2] := E_DrivingPinCtrl.Vertical;
			stError.ErrorId := pTrayTransporter^.M_ExeAction(stActionData);
			IF stError.ErrorId > 0 THEN
				nStateA_TransferTray := 99;
			ELSE
				nStateA_TransferTray := 12;
			END_IF
		END_IF
		
	12:	//TurnDrivingPin ready? -> Move slider to slot - DrivingPinGap
		IF NOT pTrayTransporter^.M_GetActionBusy(E_Action.ACTION_TurnDrivingPin) THEN
			stActionData.eAction := E_Action.ACTION_MoveTrayTransporter;
			nTransferTrayPos := pTrayTransporter^.M_GetSliderPosTrayInSlot(E_DrivingPinSelection.Right, E_TrayHollowSelection.Right) - pTrayTransporter^.P_nDrivingPinGap;
			stActionData.aParams[1] := nTransferTrayPos;
			stActionData.aParams[2] := cMoveTraySpeed;
			stError.ErrorId := pTrayTransporter^.M_ExeAction(stActionData);
			IF stError.ErrorId > 0 THEN
				nStateA_TransferTray := 99;
			ELSE
				nStateA_TransferTray := 13;
			END_IF
		END_IF
		
	13:	//Move ready? -> Move slider centre hollow (last pos - gap)
		IF NOT pTrayTransporter^.M_GetActionBusy(E_Action.ACTION_MoveTrayTransporter) THEN
			stActionData.eAction := E_Action.ACTION_MoveTrayTransporter;
			nTransferTrayPos :=  nTransferTrayPos + pTrayTransporter^.P_nDrivingPinGap;
			stActionData.aParams[1] := nTransferTrayPos;
			stActionData.aParams[2] := pTrayTransporter^.P_nMaxSliderSpeed;
			stError.ErrorId := pTrayTransporter^.M_ExeAction(stActionData);
			IF stError.ErrorId > 0 THEN
				nStateA_TransferTray := 99;
			ELSE
				nStateA_TransferTray := 14;
			END_IF
		END_IF

	14:	//Move ready? DrivingPinLeft horizontal
		IF NOT pTrayTransporter^.M_GetActionBusy(E_Action.ACTION_MoveTrayTransporter) THEN
			stActionData.eAction := E_Action.ACTION_TurnDrivingPin;
			stActionData.aParams[1] := E_DrivingPinSelection.Right;
			stActionData.aParams[2] := E_DrivingPinCtrl.Horizontal;
			stError.ErrorId := pTrayTransporter^.M_ExeAction(stActionData);
			IF stError.ErrorId > 0 THEN
				nStateA_TransferTray := 99;
			ELSE
				nStateA_TransferTray := 15;
			END_IF
		END_IF
		
	15:	//TurnDrivingPin ready? -> Lock TrayLock
		IF NOT pTrayTransporter^.M_GetActionBusy(E_Action.ACTION_TurnDrivingPin) THEN
			stActionData.eAction := E_Action.ACTION_LockUnlock;
			stActionData.aParams[1] := E_LockCtrl.Lock;
			stError.ErrorId := pTrayTransporter^.M_ExeAction(stActionData);
			IF stError.ErrorId > 0 THEN
				nStateA_TransferTray := 99;
			ELSE
				nStateA_TransferTray := 16;
			END_IF
		END_IF
		
	16:	//TrayLock ready? -> Action ready
		IF NOT pTrayTransporter^.M_GetActionBusy(E_Action.ACTION_LockUnlock) THEN
			nStateA_TransferTray := 80;
		END_IF		

END_CASE

//Errorhandling
IF nStateA_TransferTray = 99 THEN
	stError.Cmd := E_Action.ACTION_TransferTray;
	stError.POUAction := E_POUACT.POUACT_A_TransferTrayRightToSlot;
	fbErrorList.M_Add(stError);	
END_IF
END_ACTION

ACTION A_TransferTraySlotToLeft:
CASE nStateA_TransferTray OF
	0:	//TransferStation ready for transfer?
		stError.ErrorId := pTrayTransporter^.M_GetStateForTransfer(E_TransferTrayCtrl.SlotToLeft);
		IF stError.ErrorId = 0 THEN
			nStateA_TransferTray := 1;
		ELSE
			nStateA_TransferTray := 99;
		END_IF
		
	1:	//Move slider to slot
		//Hier kann es sein, dass zwei Züge erforderlich sind
		stActionData.eAction := E_Action.ACTION_MoveTrayTransporter;
		nTransferTrayPos := pTrayTransporter^.M_GetSliderPosTrayInSlot(E_DrivingPinSelection.Left, E_TrayHollowSelection.Right);
		IF nTransferTrayPos > pTrayTransporter^.P_nMaxSliderPos THEN //Mittlere Aussparung nutzen
			nTransferTrayPos := pTrayTransporter^.M_GetSliderPosTrayInSlot(E_DrivingPinSelection.Left, E_TrayHollowSelection.Centre);
			bAdditionalMoves := TRUE;
		ELSE
			bAdditionalMoves := FALSE;
		END_IF		
		stActionData.aParams[1] := nTransferTrayPos;
		stActionData.aParams[2] := pTrayTransporter^.P_nMaxSliderSpeed;
		stError.ErrorId := pTrayTransporter^.M_ExeAction(stActionData);
		IF stError.ErrorId > 0 THEN
			nStateA_TransferTray := 99;
		ELSE
			nStateA_TransferTray := 2;
		END_IF
		
	2:	//Move ready? DrivingPinLeft vertical
		IF NOT pTrayTransporter^.M_GetActionBusy(E_Action.ACTION_MoveTrayTransporter) THEN
			stActionData.eAction := E_Action.ACTION_TurnDrivingPin;
			stActionData.aParams[1] := E_DrivingPinSelection.Left;
			stActionData.aParams[2] := E_DrivingPinCtrl.Vertical;
			stError.ErrorId := pTrayTransporter^.M_ExeAction(stActionData);
			IF stError.ErrorId > 0 THEN
				nStateA_TransferTray := 99;
			ELSE
				nStateA_TransferTray := 3;
			END_IF
		END_IF
		
	3:	//TurnDrivingPin ready? -> Move slider TransferPosition left - DrivingPinGap
		IF NOT pTrayTransporter^.M_GetActionBusy(E_Action.ACTION_TurnDrivingPin) THEN
			stActionData.eAction := E_Action.ACTION_MoveTrayTransporter;
			nTransferTrayPos := pTrayTransporter^.P_nTransferPosLeft - pTrayTransporter^.P_nDrivingPinGap;
			stActionData.aParams[1] := nTransferTrayPos;
			stActionData.aParams[2] := cMoveTraySpeed;
			stError.ErrorId := pTrayTransporter^.M_ExeAction(stActionData);
			IF stError.ErrorId > 0 THEN
				nStateA_TransferTray := 99;
			ELSE
				nStateA_TransferTray := 4;
			END_IF
		END_IF
		
	4:	//Move ready? -> Move slider centre hollow (last pos + gap)
		IF NOT pTrayTransporter^.M_GetActionBusy(E_Action.ACTION_MoveTrayTransporter) THEN
			stActionData.eAction := E_Action.ACTION_MoveTrayTransporter;
			nTransferTrayPos := nTransferTrayPos + pTrayTransporter^.P_nDrivingPinGap;
			stActionData.aParams[1] := nTransferTrayPos;
			stActionData.aParams[2] := pTrayTransporter^.P_nMaxSliderSpeed;
			stError.ErrorId := pTrayTransporter^.M_ExeAction(stActionData);
			IF stError.ErrorId > 0 THEN
				nStateA_TransferTray := 99;
			ELSE
				nStateA_TransferTray := 5;
			END_IF
		END_IF
		
	5:	//Move ready? DrivingPinLeft horizontal
		IF NOT pTrayTransporter^.M_GetActionBusy(E_Action.ACTION_MoveTrayTransporter) THEN
			stActionData.eAction := E_Action.ACTION_TurnDrivingPin;
			stActionData.aParams[1] := E_DrivingPinSelection.Left;
			stActionData.aParams[2] := E_DrivingPinCtrl.Horizontal;
			stError.ErrorId := pTrayTransporter^.M_ExeAction(stActionData);
			IF stError.ErrorId > 0 THEN
				nStateA_TransferTray := 99;
			ELSE
				nStateA_TransferTray := 6;
			END_IF
		END_IF
		
	6:	//TurnDrivingPin ready? -> Move slider ??????
		//Slider muss jetzt um die Distanz von Mitte Ausssparung bis rechte Aussparung fahren
		//Achtung, Kommentar richtig stellen
		IF NOT pTrayTransporter^.M_GetActionBusy(E_Action.ACTION_TurnDrivingPin) THEN
			IF bAdditionalMoves THEN
				stActionData.eAction := E_Action.ACTION_MoveTrayTransporter;
				nTransferTrayPos := nTransferTrayPos + pTrayTransporter^.P_nTrayLength /2 - pTrayTransporter^.P_nHollowDistance;
				stActionData.aParams[1] := nTransferTrayPos;
				stActionData.aParams[2] := pTrayTransporter^.P_nMaxSliderSpeed;
				stError.ErrorId := pTrayTransporter^.M_ExeAction(stActionData);
				IF stError.ErrorId > 0 THEN
					nStateA_TransferTray := 99;
				ELSE
					nStateA_TransferTray := 7;
				END_IF
			ELSE
				nStateA_TransferTray := 11;
			END_IF
		END_IF
		
	7:	//Move ready? DrivingPinLeft vertical
		IF NOT pTrayTransporter^.M_GetActionBusy(E_Action.ACTION_MoveTrayTransporter) THEN
			stActionData.eAction := E_Action.ACTION_TurnDrivingPin;
			stActionData.aParams[1] := E_DrivingPinSelection.Left;
			stActionData.aParams[2] := E_DrivingPinCtrl.Vertical;
			stError.ErrorId := pTrayTransporter^.M_ExeAction(stActionData);
			IF stError.ErrorId > 0 THEN
				nStateA_TransferTray := 99;
			ELSE
				nStateA_TransferTray := 8;
			END_IF
		END_IF
		
	8:	//TurnDrivingPin ready? -> Move slider TransferPosLeft - DrivingPinGap
		IF NOT pTrayTransporter^.M_GetActionBusy(E_Action.ACTION_TurnDrivingPin) THEN
			stActionData.eAction := E_Action.ACTION_MoveTrayTransporter;
			nTransferTrayPos := pTrayTransporter^.P_nTransferPosLeft - pTrayTransporter^.P_nDrivingPinGap;
			stActionData.aParams[1] := nTransferTrayPos;
			stActionData.aParams[2] := pTrayTransporter^.P_nMaxSliderSpeed;
			stError.ErrorId := pTrayTransporter^.M_ExeAction(stActionData);
			IF stError.ErrorId > 0 THEN
				nStateA_TransferTray := 99;
			ELSE
				nStateA_TransferTray := 9;
			END_IF
		END_IF
		
	9:	//Move ready? -> Move slider centre hollow (last pos + gap)
		IF NOT pTrayTransporter^.M_GetActionBusy(E_Action.ACTION_MoveTrayTransporter) THEN
			stActionData.eAction := E_Action.ACTION_MoveTrayTransporter;
			nTransferTrayPos := nTransferTrayPos + pTrayTransporter^.P_nDrivingPinGap;
			stActionData.aParams[1] := nTransferTrayPos;
			stActionData.aParams[2] := pTrayTransporter^.P_nMaxSliderSpeed;
			stError.ErrorId := pTrayTransporter^.M_ExeAction(stActionData);
			IF stError.ErrorId > 0 THEN
				nStateA_TransferTray := 99;
			ELSE
				nStateA_TransferTray := 10;
			END_IF
		END_IF		
		
	10:	//Move ready? DrivingPinLeft horizontal
		IF NOT pTrayTransporter^.M_GetActionBusy(E_Action.ACTION_MoveTrayTransporter) THEN
			stActionData.eAction := E_Action.ACTION_TurnDrivingPin;
			stActionData.aParams[1] := E_DrivingPinSelection.Left;
			stActionData.aParams[2] := E_DrivingPinCtrl.Horizontal;
			stError.ErrorId := pTrayTransporter^.M_ExeAction(stActionData);
			IF stError.ErrorId > 0 THEN
				nStateA_TransferTray := 99;
			ELSE
				nStateA_TransferTray := 11;
			END_IF
		END_IF
		
	11:	//TurnDrivingPin ready? -> Move slider SafePosLeft
		IF NOT pTrayTransporter^.M_GetActionBusy(E_Action.ACTION_TurnDrivingPin) THEN
			stActionData.eAction := E_Action.ACTION_MoveTrayTransporter;
			nTransferTrayPos := pTrayTransporter^.P_nSafePosLeft;
			stActionData.aParams[1] := nTransferTrayPos;
			stActionData.aParams[2] := pTrayTransporter^.P_nMaxSliderSpeed;
			stError.ErrorId := pTrayTransporter^.M_ExeAction(stActionData);
			IF stError.ErrorId > 0 THEN
				nStateA_TransferTray := 99;
			ELSE
				nStateA_TransferTray := 12;
			END_IF
		END_IF
		
	12:	//TurnDrivingPin ready? -> Action ready
		IF NOT pTrayTransporter^.M_GetActionBusy(E_Action.ACTION_MoveTrayTransporter) THEN
			nStateA_TransferTray := 80;
		END_IF		
	
END_CASE

//Errorhandling
IF nStateA_TransferTray = 99 THEN
	stError.Cmd := E_Action.ACTION_TransferTray;
	stError.POUAction := E_POUACT.POUACT_A_TransferTraySlotToLeft;
	fbErrorList.M_Add(stError);	
END_IF
END_ACTION

ACTION A_TransferTraySlotToRight:
CASE nStateA_TransferTray OF
	0:	//TransferStation ready for transfer?
		stError.ErrorId := pTrayTransporter^.M_GetStateForTransfer(E_TransferTrayCtrl.SlotToRight);
		IF stError.ErrorId = 0 THEN
			nStateA_TransferTray := 1;
		ELSE
			nStateA_TransferTray := 99;
		END_IF
		
	1:	//Move slider to slot (right hollow with right driving pin)
		stActionData.eAction := E_Action.ACTION_MoveTrayTransporter;
		stActionData.aParams[1] := pTrayTransporter^.M_GetSliderPosTrayInSlot(E_DrivingPinSelection.Right, E_TrayHollowSelection.Right);
		stActionData.aParams[2] := pTrayTransporter^.P_nMaxSliderSpeed;
		stError.ErrorId := pTrayTransporter^.M_ExeAction(stActionData);
		IF stError.ErrorId > 0 THEN
			nStateA_TransferTray := 99;
		ELSE
			nStateA_TransferTray := 2;
		END_IF
		
	2:	//Move ready? DrivingPinLeft vertical
		IF NOT pTrayTransporter^.M_GetActionBusy(E_Action.ACTION_MoveTrayTransporter) THEN
			stActionData.eAction := E_Action.ACTION_TurnDrivingPin;
			stActionData.aParams[1] := E_DrivingPinSelection.Right;
			stActionData.aParams[2] := E_DrivingPinCtrl.Vertical;
			stError.ErrorId := pTrayTransporter^.M_ExeAction(stActionData);
			IF stError.ErrorId > 0 THEN
				nStateA_TransferTray := 99;
			ELSE
				nStateA_TransferTray := 3;
			END_IF
		END_IF
		
	3:	//Move slider TransferPosition right
		IF NOT pTrayTransporter^.M_GetActionBusy(E_Action.ACTION_TurnDrivingPin) THEN
			stActionData.eAction := E_Action.ACTION_MoveTrayTransporter;
			nTransferTrayPos := pTrayTransporter^.P_nTransferPosRight;
			stActionData.aParams[1] := nTransferTrayPos;
			stActionData.aParams[2] := cMoveTraySpeed;
			stError.ErrorId := pTrayTransporter^.M_ExeAction(stActionData);
			IF stError.ErrorId > 0 THEN
				nStateA_TransferTray := 99;
			ELSE
				nStateA_TransferTray := 4;
			END_IF		
		END_IF
		
	4:	//Move ready? -> Move slider centre hollow (last pos + gap)
		IF NOT pTrayTransporter^.M_GetActionBusy(E_Action.ACTION_MoveTrayTransporter) THEN
			stActionData.eAction := E_Action.ACTION_MoveTrayTransporter;
			nTransferTrayPos :=  nTransferTrayPos - pTrayTransporter^.P_nDrivingPinGap;
			stActionData.aParams[1] := nTransferTrayPos;
			stActionData.aParams[2] := pTrayTransporter^.P_nMaxSliderSpeed;
			stError.ErrorId := pTrayTransporter^.M_ExeAction(stActionData);
			IF stError.ErrorId > 0 THEN
				nStateA_TransferTray := 99;
			ELSE
				nStateA_TransferTray := 5;
			END_IF
		END_IF
		
	5:	//Move ready? DrivingPinRight horizontal
		IF NOT pTrayTransporter^.M_GetActionBusy(E_Action.ACTION_MoveTrayTransporter) THEN
			stActionData.eAction := E_Action.ACTION_TurnDrivingPin;
			stActionData.aParams[1] := E_DrivingPinSelection.Right;
			stActionData.aParams[2] := E_DrivingPinCtrl.Horizontal;
			stError.ErrorId := pTrayTransporter^.M_ExeAction(stActionData);
			IF stError.ErrorId > 0 THEN
				nStateA_TransferTray := 99;
			ELSE
				nStateA_TransferTray := 6;
			END_IF
		END_IF
		
	6:	//Left hollow reachable?
		IF NOT pTrayTransporter^.M_GetActionBusy(E_Action.ACTION_TurnDrivingPin) THEN
			IF bAdditionalMoves THEN
				IF nTransferTrayPos - pTrayTransporter^.P_nHollowToHollow / 2 >= pTrayTransporter^.P_nMinSliderPos THEN
					nStateA_TransferTray := 10;
				ELSE
					stError.ErrorId := E_ErrorIdCmd.ERRORID_CanNotTransferTrayCompletely;
					nStateA_TransferTray := 99; 
				END_IF
			ELSE
				IF nTransferTrayPos - pTrayTransporter^.P_nHollowToHollow >= pTrayTransporter^.P_nMinSliderPos  THEN
					nStateA_TransferTray := 10;
				ELSE
					nStateA_TransferTray := 7;
				END_IF
			END_IF
		END_IF
		
	7:	//Move slider to middle hollow
		stActionData.eAction := E_Action.ACTION_MoveTrayTransporter;
		nTransferTrayPos := nTransferTrayPos - pTrayTransporter^.P_nTrayLength/2 + pTrayTransporter^.P_nHollowDistance;
		stActionData.aParams[1] := nTransferTrayPos;
		stActionData.aParams[2] := pTrayTransporter^.P_nMaxSliderSpeed;
		stError.ErrorId := pTrayTransporter^.M_ExeAction(stActionData);
		IF stError.ErrorId > 0 THEN
			nStateA_TransferTray := 99;
		ELSE
			nStateA_TransferTray := 8;
		END_IF
		
	8:	//Move ready? DrivingPin right vertical
		IF NOT pTrayTransporter^.M_GetActionBusy(E_Action.ACTION_MoveTrayTransporter) THEN
			stActionData.eAction := E_Action.ACTION_TurnDrivingPin;
			stActionData.aParams[1] := E_DrivingPinSelection.Right;
			stActionData.aParams[2] := E_DrivingPinCtrl.Vertical;
			stError.ErrorId := pTrayTransporter^.M_ExeAction(stActionData);
			IF stError.ErrorId > 0 THEN
				nStateA_TransferTray := 99;
			ELSE
				nStateA_TransferTray := 9;
			END_IF
		END_IF
		
	9:	//TurnDrivingPin ready? -> Move TransferPosR
		IF NOT pTrayTransporter^.M_GetActionBusy(E_Action.ACTION_TurnDrivingPin) THEN
			stActionData.eAction := E_Action.ACTION_MoveTrayTransporter;
			nTransferTrayPos := pTrayTransporter^.P_nTransferPosRight;
			stActionData.aParams[1] := nTransferTrayPos;
			stActionData.aParams[2] := cMoveTraySpeed;
			stError.ErrorId := pTrayTransporter^.M_ExeAction(stActionData);
			IF stError.ErrorId > 0 THEN
				nStateA_TransferTray := 99;
			ELSE
				bAdditionalMoves := TRUE;
				nStateA_TransferTray := 4;
			END_IF
		END_IF
		
	10:	//TurnDrivingPin ready? -> Move slider at distance of both hollows (relative to previous position)
		stActionData.eAction := E_Action.ACTION_MoveTrayTransporter;
		IF bAdditionalMoves THEN //wird in State
			nTransferTrayPos := nTransferTrayPos - pTrayTransporter^.P_nHollowToHollow / 2;
		ELSE
			nTransferTrayPos := nTransferTrayPos - pTrayTransporter^.P_nHollowToHollow;	
		END_IF
		stActionData.aParams[1] := nTransferTrayPos;
		stActionData.aParams[2] := pTrayTransporter^.P_nMaxSliderSpeed;
		stError.ErrorId := pTrayTransporter^.M_ExeAction(stActionData);
		IF stError.ErrorId > 0 THEN
			nStateA_TransferTray := 99;
		ELSE
			nStateA_TransferTray := 11;
		END_IF
		
	11:	//Move ready? DrivingPinRight vertical
		IF NOT pTrayTransporter^.M_GetActionBusy(E_Action.ACTION_MoveTrayTransporter) THEN
			stActionData.eAction := E_Action.ACTION_TurnDrivingPin;
			stActionData.aParams[1] := E_DrivingPinSelection.Right;
			stActionData.aParams[2] := E_DrivingPinCtrl.Vertical;
			stError.ErrorId := pTrayTransporter^.M_ExeAction(stActionData);
			IF stError.ErrorId > 0 THEN
				nStateA_TransferTray := 99;
			ELSE
				nStateA_TransferTray := 12;
			END_IF
		END_IF
		
	12:	//TurnDrivingPin ready? -> Move TransferPosR + DrivingPinGap
		IF NOT pTrayTransporter^.M_GetActionBusy(E_Action.ACTION_TurnDrivingPin) THEN
			stActionData.eAction := E_Action.ACTION_MoveTrayTransporter;
			nTransferTrayPos := pTrayTransporter^.P_nTransferPosRight + pTrayTransporter^.P_nDrivingPinGap;
			stActionData.aParams[1] := nTransferTrayPos;
			stActionData.aParams[2] := cMoveTraySpeed;
			stError.ErrorId := pTrayTransporter^.M_ExeAction(stActionData);
			IF stError.ErrorId > 0 THEN
				nStateA_TransferTray := 99;
			ELSE
				nStateA_TransferTray := 13;
			END_IF
		END_IF
		
	13:	//Move ready? -> Move slider centre hollow (last pos + gap)
		IF NOT pTrayTransporter^.M_GetActionBusy(E_Action.ACTION_MoveTrayTransporter) THEN
			stActionData.eAction := E_Action.ACTION_MoveTrayTransporter;
			nTransferTrayPos :=  nTransferTrayPos - pTrayTransporter^.P_nDrivingPinGap;
			stActionData.aParams[1] := nTransferTrayPos;
			stActionData.aParams[2] := pTrayTransporter^.P_nMaxSliderSpeed;
			stError.ErrorId := pTrayTransporter^.M_ExeAction(stActionData);
			IF stError.ErrorId > 0 THEN
				nStateA_TransferTray := 99;
			ELSE
				nStateA_TransferTray := 14;
			END_IF
		END_IF
		
	14:	//Move ready? DrivingPinRight horizontal
		IF NOT pTrayTransporter^.M_GetActionBusy(E_Action.ACTION_MoveTrayTransporter) THEN
			stActionData.eAction := E_Action.ACTION_TurnDrivingPin;
			stActionData.aParams[1] := E_DrivingPinSelection.Right;
			stActionData.aParams[2] := E_DrivingPinCtrl.Horizontal;
			stError.ErrorId := pTrayTransporter^.M_ExeAction(stActionData);
			IF stError.ErrorId > 0 THEN
				nStateA_TransferTray := 99;
			ELSE
				nStateA_TransferTray := 15;
			END_IF
		END_IF
		
	15:	//TurnDrivingPin ready? -> Action ready
		IF NOT pTrayTransporter^.M_GetActionBusy(E_Action.ACTION_TurnDrivingPin) THEN
			nStateA_TransferTray := 80;
		END_IF		
		
END_CASE

//Errorhandling
IF nStateA_TransferTray = 99 THEN
	stError.Cmd := E_Action.ACTION_TransferTray;
	stError.POUAction := E_POUACT.POUACT_A_TransferTraySlotToRight;
	fbErrorList.M_Add(stError);	
END_IF
END_ACTION

ACTION A_WashTool:
stError.POUState := nActionState;

IF pMzTool^.P_bError THEN
	stError.ObjectId := pMzTool^.P_nObjectID;
	stError.ErrorId := pMzTool^.P_nErrorId;
	nActionState := 99;	
ELSIF pWashStation^.P_bError THEN
	stError.ObjectId := pWashStation^.P_nObjectID;
	stError.ErrorId := pWashStation^.P_nErrorId;
	nActionState := 99;
END_IF

CASE nActionState OF
	0:	//MoveToTarget "Washpoint"
		MEMSET(ADR(stActionData),0,SIZEOF(stActionData));
		stActionData.eAction := E_Action.ACTION_MoveToTarget;
		IF pMzTool^.P_eObjectType = E_ObjectType.OBJECTTYPE_TwinPiezoHolder THEN
			pTwinPiezoHolder := pMzTool;
 			stActionData.nObject := pTwinPiezoHolder^.P_pPiezoPipFirst^.P_nObjectID;
		ELSE
			stActionData.nObject := pMzTool^.P_nObjectID;
		END_IF
		
		stActionData.nTarget := pTarget^.P_nObjectID;
		stActionData.aParams[1] := E_TargetRef.TARGETREF_SpecPoint;
		stActionData.aParams[2] := nSpecPointSlotNr;
		stActionData.aParams[5] := -1;	//MaxSpeed X
		stActionData.aParams[6] := -1;	//MaxSpeed Y
		stActionData.aParams[7] := -1;	//Speed Z
		
		stError.ErrorId := fbMoveToTarget.M_SetAndCheckParams(stActionData);
		IF stError.ErrorId > 0 THEN	//Error
			nActionState := 99;
		ELSE
			fbMoveToTarget(bExecute:= TRUE);
			nActionState := 1;
		END_IF
		
	1:	//MoveToTarget ready?
		fbMoveToTarget(bExecute:= TRUE);
		IF NOT fbMoveToTarget.bBusy THEN
			IF fbMoveToTarget.bError THEN
				stError.ErrorId := fbMoveToTarget.nErrorId;
				nActionState := 99;
			ELSE
				nActionState := 2;
				//WastePumpe in jedem Fall einschalten
				IF eWashMode <> E_WashMode.MODE_DryOutside THEN
					MEMSET(ADR(stActionData),0,SIZEOF(stActionData));
					stActionData.eAction := E_Action.ACTION_SwitchPump;
					stActionData.aParams[1] := 0; //WastePump
					stActionData.aParams[2] := 1; //On
					stError.ErrorId := pWashStation^.M_ExeAction(stActionData);
					IF stError.ErrorId > 0 THEN
						nActionState := 99;
					END_IF
				END_IF
			END_IF
			fbMoveToTarget(bExecute:= FALSE);
		END_IF
		
	2:	//Abhängig vom Washmode Dispensen bzw. Washststation aktivieren
		nActionState := 3;
		MEMSET(ADR(stActionData),0,SIZEOF(stActionData));
		CASE eWashMode OF
			E_WashMode.MODE_WashInside:
				//Tool dispensen
				//Für den Fall, dass Tool eine Piezo ist, dann soll diese auch Dispense Drops ausführen
				stActionData.eAction := E_Action.ACTION_Dispense;
				//überprüfen, ob bei nQuantity 0, ein Dauerdispensen erfolgt.
				//bisher noch nicht, es wurde nur beim HybridDispenser benutzt
				//es kann aber noch in M_ExeAction so umgebaut werden, dass es so funktioniert.
				stActionData.aParams[1] := nQuantity1;
				stActionData.aParams[2] := nFlow1;
				stActionData.aParams[3] := nDilInputNr;
				stError.ErrorId := pMzTool^.M_ExeAction(stActionData);
				IF stError.ErrorId = 0 THEN
					//Für den Fall, dass Tool eine Piezo ist, dann soll diese auch Dispense Drops machen ausführen
					IF pMzTool^.P_eObjectType = E_ObjectType.OBJECTTYPE_PiezoPip OR pMzTool^.P_eObjectType = E_ObjectType.OBJECTTYPE_TwinPiezoHolder THEN
						MEMSET(ADR(stActionData),0,SIZEOF(stActionData));
						stActionData.eAction := E_Action.ACTION_DispenseDrops;
						stActionData.aParams[2] := 1; //DispCtrl = On
						stActionData.aParams[5] := 1; //Skip valve move
						stError.ErrorId := pMzTool^.M_ExeAction(stActionData);
					END_IF
				END_IF
				nActionState := 3;
			E_WashMode.MODE_WashInOutside:
				//Washstation spülen Ein
				stActionData.eAction := E_Action.ACTION_Rinse;
				stActionData.aParams[1] := nRinseChannel;
				stActionData.aParams[2] := 1; //Rinse "ON
				stActionData.aParams[3] := DWORD_TO_DINT(nTime); //Time
				stActionData.aParams[4] := 1; //KeepWastePumpOn
				stError.ErrorId := pWashStation^.M_ExeAction(stActionData);
				IF stError.ErrorId = 0 THEN
					stActionData.eAction := E_Action.ACTION_Dispense;
					stActionData.aParams[1] := nQuantity1;
					stActionData.aParams[2] := nFlow1;
					stActionData.aParams[3] := nDilInputNr;
					stError.ErrorId := pMzTool^.M_ExeAction(stActionData);
					IF stError.ErrorId = 0 THEN
						//Für den Fall, dass Tool eine Piezo ist, dann soll diese auch Dispense Drops machen ausführen
						IF pMzTool^.P_eObjectType = E_ObjectType.OBJECTTYPE_PiezoPip OR pMzTool^.P_eObjectType = E_ObjectType.OBJECTTYPE_TwinPiezoHolder THEN
							MEMSET(ADR(stActionData),0,SIZEOF(stActionData));
							stActionData.eAction := E_Action.ACTION_DispenseDrops;
							stActionData.aParams[2] := 1; //DispCtrl = On
							stActionData.aParams[5] := 1; //Skip valve move
							stError.ErrorId := pMzTool^.M_ExeAction(stActionData);
						END_IF
					END_IF
					nActionState := 3;
				END_IF
			E_WashMode.MODE_WashOutside:
				//Washstation spülen Ein
				stActionData.eAction := E_Action.ACTION_Rinse;
				stActionData.aParams[1] := nRinseChannel;
				stActionData.aParams[2] := 1; //Rinse "ON
				stActionData.aParams[3] := UDINT_TO_DINT(nTime); //Time
				stError.ErrorId := pWashStation^.M_ExeAction(stActionData);
				nActionState := 3;
			E_WashMode.MODE_DryOutside:
				//Luftdusche "Ein"
				stError.ErrorId := pWashStation^.M_SwitchAirShower(TRUE);
				nActionState := 10;
		END_CASE
		
		IF stError.ErrorId > 0 THEN
			nActionState := 99;
		END_IF					
		
	3:	//warten bis Dispensen bzw Time abgelaufen
		CASE eWashMode OF
			E_WashMode.MODE_WashInside:
				//Warten, bis Dispensen fertig
				IF NOT pMzTool^.M_GetActionBusy(E_ACTION.ACTION_Dispense) THEN
					pMzTool^.M_CancelAction(E_Action.ACTION_DispenseDrops);
					//WashStation leeren (dadurch wird aktivierte Wastepumpe auch abgeschalten)
					stActionData.eAction := E_Action.ACTION_EmptyWaste;
					pWashStation^.M_ExeAction(stActionData);
					nActionState := 4; //langsam heraus fahren
				END_IF
			E_WashMode.MODE_WashInOutside:
				//Für den Fall, dass Dispense auf Dauerdispensen eingestellt ist dann muss dieses abgebrochen werden wenn Rinse
				//fertig ist.
				IF nQuantity1 = 0 THEN //Dauerdispensen
					IF NOT pWashStation^.M_GetActionBusy(E_ACTION.ACTION_Rinse) THEN
						pMzTool^.M_CancelAction(E_Action.ACTION_Dispense);
						pMzTool^.M_CancelAction(E_Action.ACTION_DispenseDrops);
						//WashStation leeren (dadurch wird aktivierte Wastepumpe auch abgeschalten)
						stActionData.eAction := E_Action.ACTION_EmptyWaste;
						pWashStation^.M_ExeAction(stActionData);
						nActionState := 4; //langsam heraus fahren
					END_IF
				ELSE
					IF NOT (pMzTool^.M_GetActionBusy(E_ACTION.ACTION_Dispense) OR pWashStation^.M_GetActionBusy(E_ACTION.ACTION_Rinse)) THEN
						pMzTool^.M_CancelAction(E_Action.ACTION_DispenseDrops);
						//WashStation leeren (dadurch wird aktivierte Wastepumpe auch abgeschalten)
						stActionData.eAction := E_Action.ACTION_EmptyWaste;
						pWashStation^.M_ExeAction(stActionData);
						nActionState := 4; //langsam heraus fahren
					END_IF					
				END_IF
			E_WashMode.MODE_WashOutside:
				IF NOT pWashStation^.M_GetActionBusy(E_ACTION.ACTION_Rinse) THEN
					nActionState := 6; //Move free
				END_IF			
		END_CASE
		
	4:	//MoveZ bis OK WashStation langsam
		MEMSET(ADR(stActionData),0,SIZEOF(stActionData));
		stActionData.eAction := E_Action.ACTION_MoveZ;
		stActionData.aParams[1] := E_MoveMode.MODE_AbsWithOffset;
		stPoint1 := pWashStation^.P_stAbsPosCenter;
		stActionData.aParams[2] := REAL_TO_DINT(stPoint1.Z);
		stActionData.aParams[3] := 5000; //Speed
		stError.ErrorId := pMzTool^.M_ExeAction(stActionData);
		IF stError.ErrorId > 0 THEN
			nActionState := 99;
		ELSE
			nActionState := 5;
		END_IF
		
	5:	//MoveZ ready?
		IF NOT pMzTool^.M_GetActionBusy(E_Action.ACTION_MoveZ) THEN
			nActionState := 6;
		END_IF
	
	6:	//MoveFree
		MEMSET(ADR(stActionData),0,SIZEOF(stActionData));
		stActionData.eAction := E_Action.ACTION_MoveZ;
		stActionData.aParams[1] := E_MoveMode.MODE_Free;
		stActionData.aParams[3] := -1;	//MaxSpeed
		stError.ErrorId := pMzTool^.M_ExeAction(stActionData);
		IF stError.ErrorId > 0 THEN	//Error
			nActionState := 99;
		ELSE
			nActionState := 7;
		END_IF
		
	7:	//MoveFree ready?
		IF NOT pMzTool^.M_GetActionBusy(E_Action.ACTION_MoveZ) THEN
			nActionState := 80;
		END_IF

	10:	//Drying
		//MoveUp über Zeit
		//Distance berechnen aus aktueller Position minus Oberkante WashStation
		//Speed berechnen aus Distance und Time
		//Achtung! Begrenzung MaxSpeed
		stPoint1 := pMzTool^.P_stCurrentPosTotal;
		stPoint2 := pWashStation^.P_stAbsPosCenter;
		MEMSET(ADR(stActionData),0,SIZEOF(stActionData));
		stActionData.eAction := E_Action.ACTION_MoveZ;
		stActionData.aParams[1] := E_MoveMode.MODE_AbsWithOffset;
		stActionData.aParams[2] := REAL_TO_DINT(stPoint2.Z); //Oberkante Waschstation
		stActionData.aParams[3] :=  REAL_TO_DINT((stPoint2.Z - stPoint1.Z) / (UDINT_TO_REAL(nTime) / 1000.0)); //Speed berechnet aus Zeit und Weg
		stError.ErrorId := pMzTool^.M_ExeAction(stActionData);
		IF stError.ErrorId > 0 THEN	//Error
			nActionState := 99;
		ELSE
			nActionState := 11;
		END_IF
		
	11:	//MoveUp ready?
		IF NOT pMzTool^.M_GetActionBusy(E_Action.ACTION_MoveZ) THEN
			pWashStation^.M_SwitchAirShower(FALSE);
			nActionState := 4;
		END_IF
	
	70:	//Abbrechen
		nActionState := 80;
		//Actionen der beteiligten Decvices abbrechen
		//MoveToTarget oder MoveZ vom MzTool abbrechen (schließen sich gegenseitig aus)
		IF fbMoveToTarget.bBusy THEN
			nActionState := 70;
			fbMoveToTarget(bStop:= TRUE);
		ELSIF pMzTool^.M_GetActionBusy(E_Action.ACTION_MoveZ) THEN
			nActionState := 70;
			pMzTool^.M_CancelAction(E_Action.ACTION_MoveZ);
		ELSE
			fbMoveToTarget(bExecute:= FALSE);
		END_IF
		
		IF pMzTool^.M_GetActionBusy(E_Action.ACTION_Dispense) THEN
			nActionState := 70;
			pMzTool^.M_CancelAction(E_Action.ACTION_Dispense);
		END_IF
		
		IF pMzTool^.M_GetActionBusy(E_Action.ACTION_DispenseDrops) THEN
			nActionState := 70;
			pMzTool^.M_CancelAction(E_Action.ACTION_DispenseDrops);
		END_IF

		IF pMzTool^.M_GetActionBusy(E_Action.ACTION_SetPressure) THEN
			nActionState := 70;
			pMzTool^.M_CancelAction(E_Action.ACTION_SetPressure);
		END_IF
		
		IF pMzTool^.M_GetActionBusy(E_Action.ACTION_SwitchPressure) THEN
			nActionState := 70;
			pMzTool^.M_CancelAction(E_Action.ACTION_SwitchPressure);
		END_IF
		
		pWashStation^.M_Stop();	
END_CASE

//Errorhandling
IF nActionState = 99 THEN
	pMzTool^.M_Stop();
	pWashStation^.M_Stop();
	fbMoveToTarget(bExecute:= FALSE);
	stError.Cmd := E_Action.ACTION_WashTool;
	stError.POUAction := E_POUACT.POUACT_A_WashTool;
	fbErrorList.M_Add(stError);	
END_IF
END_ACTION

METHOD FB_init : BOOL
VAR_INPUT
	bInitRetains : BOOL; // if TRUE, the retain variables are initialized (warm start / cold start)
	bInCopyCode : BOOL;  // if TRUE, the instance afterwards gets moved into the copy code (online change)
END_VAR
stError.POU := E_POU.POU_FB_ComplexAction;
END_METHOD

METHOD M_Continue
VAR_INPUT
END_VAR
IF eCurrentState = E_MachineState.MACHINESTATE_Pause THEN
	eCurrentState := E_MachineState.MACHINESTATE_Active;
END_IF
END_METHOD

METHOD M_ExeAction : ERRORID
VAR_INPUT
	refActionData : REFERENCE TO ST_ActionData;
END_VAR

VAR
	i			: UINT;
	nObjectId	: UINT;
END_VAR
VAR CONSTANT
	cHighVoltThreshold : DINT := 25;
END_VAR
//Es kann immer nur eine ComplexAction aktiv werden
IF eCurrentState = E_MachineState.MACHINESTATE_Active THEN
	M_ExeAction := E_ErrorIdCmd.ERRORID_ComplexActionActive;
	RETURN;
END_IF

IF eCurrentState = E_MachineState.MACHINESTATE_PauseRequest OR eCurrentState = E_MachineState.MACHINESTATE_Pause THEN
	M_ExeAction := E_ErrorIdCmd.ERRORID_ComplexActionActive;
	RETURN;
END_IF

IF NOT eCurrentState = E_MachineState.MACHINESTATE_Idle THEN
	M_ExeAction := E_ErrorIdCmd.ERRORID_InvalidState;
	RETURN;	
END_IF

//Es darf keine XY-Bewegung an einem Kopf stattfinden (mit Ausnahme)
//Welche Ausnahme soll denn das sein?
FOR i:= 1 TO fbObjectDirectory.nCntMZHead BY 1 DO 
	IF afbMzHead[i].P_bZIsMoving OR afbMzHead[i].P_bXYIsMoving THEN
		M_ExeAction := E_ErrorIdMultiZ.ERRORID_MultiZIsStillMoving;
		RETURN;
	END_IF
END_FOR

CASE refActionData.eAction OF
	E_Action.ACTION_ActionOnArray:
		//Object gültiges MzTool?
		IF fbObjectDirectory.M_ObjIsMzTool(refActionData.nObject) THEN
			pMzTool := fbObjectDirectory.M_GetObjPointer(refActionData.nObject);
		ELSE 
			M_ExeAction := E_ErrorIdCmd.ERRORID_UnsuitableObject;  //Error
			RETURN;
		END_IF
		
		eActOnArrayOrder := DINT_TO_USINT(refActionData.aParams[1]);
		nActOnArraySpeedX := refActionData.aParams[2];
		nActOnArraySpeedY := refActionData.aParams[3];
		nActOnArraySpeedZ := refActionData.aParams[4];
		nActOnArraySpeedZRelease := refActionData.aParams[5];
		nZOffset1 := refActionData.aParams[6];	//ZOffsetAction
		nDistance1 := refActionData.aParams[7];	//ZDistanceRelease
		nZOffset2 := refActionData.aParams[8];	//ZOffsetXYMove
		
		bReleaseMoveInstantly := DINT_TO_BOOL(refActionData.aParams[9]);
		tReleaseMoveDelay := DINT_TO_TIME(refActionData.aParams[10]);
		
		//SubAction von stActionData auf stActionData2 übertragen
		
		MEMSET(ADR(stActionData2),0,SIZEOF(stActionData2));
		stActionData2.nObject := refActionData.nObject;
		stActionData2.eAction := DINT_TO_UINT(refActionData.aParams[11]);
		MEMCPY(ADR(stActionData2.aParams),ADR(refActionData.aParams[12]),32);
		
		
		//Action mit MzTool ausführbar?
		M_ExeAction := pMzTool^.M_CheckAction(stActionData2,0); 
		IF M_ExeAction > 0 THEN //Error
			RETURN;
		END_IF
		
		//Ist die Action im Allgemeinen geeignet?
		IF NOT(stActionData2.eAction = E_Action.ACTION_Aspirate OR
			stActionData2.eAction = E_Action.ACTION_Dispense OR
			stActionData2.eAction = E_Action.ACTION_DispenseDrops OR
			stActionData2.eAction = E_Action.ACTION_Expose OR
			stActionData2.eAction = E_Action.ACTION_Extrude OR
			stActionData2.eAction = E_Action.ACTION_PickPutPowder OR
			stActionData2.eAction = E_Action.ACTION_PulsePressure OR
			stActionData2.eAction = E_Action.ACTION_StampDemolding OR
			stActionData2.eAction = E_Action.ACTION_Mix OR
			stActionData2.eAction = E_Action.ACTION_SwitchPressure OR
			stActionData2.eAction = E_Action.ACTION_TakePicture) THEN
			M_ExeAction := E_ErrorIdCmd.ERRORID_InvalidAction;
			RETURN;
		END_IF
		
		IF fbObjectDirectory.M_GetObjType(refActionData.nTarget) = E_ObjectType.OBJECTTYPE_SpotArray OR
			fbObjectDirectory.M_GetObjType(refActionData.nTarget) = E_ObjectType.OBJECTTYPE_Mtp THEN
			pTarget := fbObjectDirectory.M_GetObjPointer(refActionData.nTarget);
			pArray := pTarget;
			nTargetCol := 0;
			nTargetRow := 0;
		ELSE
			M_ExeAction := E_ErrorIdCmd.ERRORID_UnsuitableTarget;  //Error
			RETURN;
		END_IF
		
		pHighVoltTray := pTarget^.M_GetFirstParentOfType(E_ObjectType.OBJECTTYPE_HighVoltTray);
		IF pHighVoltTray > 0 THEN
			IF pMzTool^.P_eObjectType = E_ObjectType.OBJECTTYPE_CartDispenser OR 
									pMzTool^.P_eObjectType = E_ObjectType.OBJECTTYPE_CartDispStirrer THEN
				pCartDispenser := pMzTool;
			END_IF			
			IF pHighVoltTray^.P_nCurrentVoltage > cHighVoltThreshold THEN
				IF NOT(pCartDispenser > 0 AND_THEN pCartDispenser^.P_bIsMESTool) THEN
					M_ExeAction := E_ErrorIdCmd.ERRORID_RiskHighvoltFlashover;
					RETURN;
				END_IF
			END_IF
		END_IF
		
	E_Action.ACTION_CalibrateZSensor:
		IF fbObjectDirectory.M_GetObjType(refActionData.nObject) = E_ObjectType.OBJECTTYPE_ZSensor THEN
			pZLevelSensor := fbObjectDirectory.M_GetObjPointer(refActionData.nObject);
			pTarget := fbObjectDirectory.M_GetObjPointer(refActionData.nTarget);
			//ZSensor montiert?
			IF NOT pZLevelSensor^.P_bSensorMounted THEN
				M_ExeAction := E_ErrorIdCmd.ERRORID_ZSensorNotMounted;  //Error
				RETURN;
			END_IF
			//ZSensor kann nur an einem "Point" kalibriert werden
			IF fbObjectDirectory.M_GetObjType(refActionData.nTarget) <> E_ObjectType.OBJECTTYPE_Point THEN
				M_ExeAction := E_ErrorIdCmd.ERRORID_UnsuitableTarget; //Error
				RETURN;	
			END_IF
			//Point darf keinen Offset haben
			IF pTarget^.P_rZOffset <> 0.0 THEN
				M_ExeAction := E_ErrorIdCmd.ERRORID_CalibrationPointHasAnOffset; //Error
				RETURN;	
			END_IF
		ELSE
			M_ExeAction := E_ErrorIdCmd.ERRORID_UnsuitableObject; //Error
			RETURN;
		END_IF

		pHighVoltTray := pTarget^.M_GetFirstParentOfType(E_ObjectType.OBJECTTYPE_HighVoltTray);
		IF pHighVoltTray > 0 THEN
			IF pHighVoltTray^.P_nCurrentVoltage > cHighVoltThreshold THEN
				M_ExeAction := E_ErrorIdCmd.ERRORID_RiskHighvoltFlashover;
				RETURN;
			END_IF
		END_IF
	
	E_Action.ACTION_CleanTip:
		//Mit Object ausführbar?
		pMzTool := fbObjectDirectory.M_GetObjPointer(refActionData.nObject);
		IF pMzTool = 0 THEN
			M_ExeAction := E_ErrorIdCmd.ERRORID_UnsuitableObject;
			RETURN;
		END_IF
		
		CASE pMzTool^.P_eObjectType OF
			E_ObjectType.OBJECTTYPE_CartDispenser,
			E_ObjectType.OBJECTTYPE_CartDispStirrer:
				pCartDispenser := pMzTool;
				iDispenser := pCartDispenser^;
			E_ObjectType.OBJECTTYPE_MultiCartHolder:
				pMultiCartHolder := pMzTool;
				iDispenser := pMultiCartHolder^;
			E_ObjectType.OBJECTTYPE_Extruder:
				pExtruder := pMzTool;
				iDispenser := pExtruder^;
			E_ObjectType.OBJECTTYPE_TwinExtruder:
				pTwinExtruder := pMzTool;
				iDispenser := pTwinExtruder^;
			E_ObjectType.OBJECTTYPE_HybridDispenser:
				pHybridDispenser := pMzTool;
				iDispenser := pHybridDispenser^;
			E_ObjectType.OBJECTTYPE_PassivPip:
				pPassivePip := pMzTool;
				iDispenser := pPassivePip^;
		ELSE
			M_ExeAction := E_ErrorIdCmd.ERRORID_UnsuitableObject;
			RETURN;
		END_CASE
		
		pTipCleaner := 0;
		pTipCleanerGen2 := 0;
		//Ist Target ein TipCleaner?
		CASE fbObjectDirectory.M_GetObjType(refActionData.nTarget)OF
			E_ObjectType.OBJECTTYPE_TipCleaner:
				pTipCleaner := fbObjectDirectory.M_GetObjPointer(refActionData.nTarget);
			E_ObjectType.OBJECTTYPE_TipCleanerGen2:
				pTipCleaner := fbObjectDirectory.M_GetObjPointer(refActionData.nTarget);
				pTipCleanerGen2 := pTipCleaner;
				pSlot := pTipCleanerGen2^.M_GetSlot(DINT_TO_UINT(refActionData.aParams[1]));
				IF pSlot = 0 THEN
					M_ExeAction := E_ErrorIdCmd.ERRORID_InvalidTargetSlot;
					RETURN;
				END_IF
				eCleaningMode := DINT_TO_USINT(refActionData.aParams[2]);
				tCleaningDispenseTime := DINT_TO_TIME(refActionData.aParams[3]);
				nCleaningWireSpeed := refActionData.aParams[4];
				IF nCleaningWireSpeed < 1 THEN
					M_ExeAction := E_ErrorIdCmd.ERRORID_InvalidCleaningWireSpeed;
					RETURN;
				END_IF
		ELSE
			M_ExeAction := E_ErrorIdCmd.ERRORID_UnsuitableTarget;
			RETURN;
		END_CASE
 		
		
	E_Action.ACTION_DispenseTest:
		IF (fbObjectDirectory.M_GetObjType(refActionData.nObject) <> E_ObjectType.OBJECTTYPE_PiezoPip) AND
			(fbObjectDirectory.M_GetObjType(refActionData.nObject) <> E_ObjectType.OBJECTTYPE_TwinPiezoHolder) THEN //Object gültiges MzTool?
			M_ExeAction := E_ErrorIdCmd.ERRORID_UnsuitableObject;
			RETURN;
		END_IF

		IF fbObjectDirectory.M_GetObjType(refActionData.nTarget) <> E_ObjectType.OBJECTTYPE_Stroboscope THEN //Target gültig?
			M_ExeAction := E_ErrorIdCmd.ERRORID_UnsuitableTarget;
			RETURN;
		END_IF	
		
		pMzTool := fbObjectDirectory.M_GetObjPointer(refActionData.nObject);
		pPiezoPip := pMzTool;
		pStroboscope := fbObjectDirectory.M_GetObjPointer(refActionData.nTarget);
		nDispenseTestArg2 := refActionData.aParams[1];
		bInhibitDispenseTrials := DINT_TO_BOOL(refActionData.aParams[2]);
		
	E_Action.ACTION_DockTool:
		IF fbObjectDirectory.M_ObjIsMzTool(refActionData.nObject) THEN //Gültiges MzTool?
			pMzTool := fbObjectDirectory.M_GetObjPointer(refActionData.nObject);
		ELSE 
			M_ExeAction := E_ErrorIdCmd.ERRORID_UnsuitableObject;  //Error
			RETURN;
		END_IF
		
		IF fbObjectDirectory.M_ObjIsTarget(refActionData.nTarget) THEN //Gültiges Target?
			pTarget := fbObjectDirectory.M_GetObjPointer(refActionData.nTarget);
		ELSE
			M_ExeAction := E_ErrorIdCmd.ERRORID_UnsuitableTarget;  //Error
			RETURN;
		END_IF
		
		M_ExeAction := pMzTool^.M_CheckAction(refActionData,pTarget); //Ausführbar mit MzTool?
		IF M_ExeAction > 0 THEN
			RETURN;
		END_IF
		
		M_ExeAction := pTarget^.M_CheckAction(refActionData,pMzTool); //Ausführbar mit Target?
		IF M_ExeAction > 0 THEN
			RETURN;
		END_IF
		
		IF pMzTool^.P_eObjectType = E_ObjectType.OBJECTTYPE_Luer THEN
			pLuer := pMzTool;
			rSumDockOffset := pLuer^.P_rDockOffset;
		ELSIF pMzTool^.P_eObjectType = E_ObjectType.OBJECTTYPE_TriplePip THEN
			pTriplePip := pMzTool;
			rSumDockOffset := pTriplePip^.P_rDockOffset;
		ELSIF pMzTool^.P_eObjectType = E_ObjectType.OBJECTTYPE_VacuumHandler THEN
			pVacuumHandler := pMzTool;
			rSumDockOffset := pVacuumHandler^.P_rDockOffset;
		ELSE
			rSumDockOffset := 0;
		END_IF
		
		IF (pTarget^.P_eObjectGroup AND E_ObjectGroup.OBJECTGROUP_Rack) = E_ObjectGroup.OBJECTGROUP_Rack THEN
			pRack := pTarget;
			pPieceSlot := pRack^.M_GetSlot(DINT_TO_UINT(refActionData.aParams[2]));
		ELSIF pTarget^.P_eObjectType = E_ObjectType.OBJECTTYPE_Reactor THEN
			pReactor := pTarget;
			pPieceSlot := pReactor^.M_GetSlot(1);
		END_IF
		
		IF pPieceSlot > 0 THEN
			IF pPieceSlot^.P_pPiece > 0 THEN
				rSumDockOffset := rSumDockOffset + pPieceSlot^.P_pPiece^.P_rDockOffset;
			END_IF
		END_IF
		
		nZOffset1 := refActionData.aParams[4];
		
	E_Action.ACTION_DryPip:
		//Object gültiges MzTool?
		IF fbObjectDirectory.M_ObjIsMzTool(refActionData.nObject) THEN
			pMzTool := fbObjectDirectory.M_GetObjPointer(refActionData.nObject);
		ELSE 
			M_ExeAction := E_ErrorIdCmd.ERRORID_UnsuitableObject;  //Error
			RETURN;
		END_IF

		//Ist Target ein Drypad
		IF fbObjectDirectory.M_GetObjType(refActionData.nTarget) <> E_ObjectType.OBJECTTYPE_DryPad THEN
			M_ExeAction := E_ErrorIdCmd.ERRORID_UnsuitableTarget;
			RETURN;
		END_IF
		
		pDryPad := fbObjectDirectory.M_GetObjPointer(refActionData.nTarget);

		CASE pMzTool^.P_eObjectType OF
			E_ObjectType.OBJECTTYPE_PassivPip:
				pPassivePip := pMzTool;
				iUsingDryPad := pPassivePip^;
			E_ObjectType.OBJECTTYPE_PiezoPip:
				pPiezoPip := pMzTool;
				iUsingDryPad := pPiezoPip^;
			E_ObjectType.OBJECTTYPE_SolenoidPip:
				pSolenoidPip := pMzTool;
				iUsingDryPad := pSolenoidPip^;
			E_ObjectType.OBJECTTYPE_TwinPiezoHolder:
				pTwinPiezoHolder := pMzTool;
				IF (pTwinPiezoHolder^.P_pPiezoPipFirst = 0) OR (pTwinPiezoHolder^.P_pPiezoPipSecond = 0) THEN
					M_ExeAction := E_ErrorIdCmd.ERRORID_NotAllPipettesConfigured;
					RETURN;
				ELSE
					iUsingDryPad := pTwinPiezoHolder^.P_pPiezoPipFirst^;
					pMzTool := pTwinPiezoHolder^.P_pPiezoPipFirst;
				END_IF
			E_ObjectType.OBJECTTYPE_Luer:
				//Luer kann derzeit nur mit Needle oder Tip auf dem DryPad trocknen (Kollision)
				IF pMzTool^.P_pPiece = 0 THEN
					M_ExeAction := E_ErrorIdCmd.ERRORID_NoPieceOnTool; //Error
					RETURN;
				END_IF
				pLuer :=  pMzTool;
				iUsingDryPad := pLuer^;
		ELSE
			M_ExeAction := E_ErrorIdCmd.ERRORID_InvalidAction;  //Error
			RETURN;
		END_CASE

		IF refActionData.aParams[1] > 0 THEN
			nTime := DINT_TO_UDINT(refActionData.aParams[1]);
		ELSE
			nTime := TIME_TO_UDINT(iUsingDryPad.P_tDryTime);
		END_IF
		nZOffset1 := refActionData.aParams[2];
		
	E_Action.ACTION_DryToolInside:
		IF fbObjectDirectory.M_ObjIsMzTool(refActionData.nObject) THEN //Gültiges MzTool?
			pMzTool := fbObjectDirectory.M_GetObjPointer(refActionData.nObject);
		ELSE 
			M_ExeAction := E_ErrorIdCmd.ERRORID_UnsuitableObject;  //Error
			RETURN;
		END_IF	
		
		IF fbObjectDirectory.M_GetObjType(refActionData.nTarget) <> E_ObjectType.OBJECTTYPE_WashStation THEN //gültiges Target?
			M_ExeAction := E_ErrorIdCmd.ERRORID_UnsuitableTarget;
			RETURN;
		ELSE
			pWashStation := fbObjectDirectory.M_GetObjPointer(refActionData.nTarget);
		END_IF
		
		//Kann Tool Action ausführen?
		M_ExeAction := pMzTool^.M_CheckAction(refActionData, pWashStation);
		IF M_ExeAction > 0 THEN
			RETURN;
		END_IF
		
		//Kann WashStation Action ausführen?
		M_ExeAction := pWashStation^.M_CheckAction(refActionData, pMzTool);
		IF M_ExeAction > 0 THEN
			RETURN;
		END_IF
		
		nSpecPointSlotNr := DINT_TO_UINT(refActionData.aParams[1]);
		nPressure1 := DINT_TO_INT(refActionData.aParams[2]);
		nTime := DINT_TO_DWORD(refActionData.aParams[3]);

	E_Action.ACTION_ExchangePiece:
		IF refActionData.aParams[2] = 0 THEN
			bTakePiece := FALSE;
		ELSIF refActionData.aParams[2] = 1 THEN
			bTakePiece := TRUE;
		ELSE
			M_ExeAction := E_ErrorIdCmd.ERRORID_InvalidCtrl;
			RETURN;
		END_IF
		
		eExchangeOption := DINT_TO_USINT(refActionData.aParams[3]);
		
		IF NOT (eExchangeOption = E_ExchangePieceOption.Slot OR eExchangeOption = E_ExchangePieceOption.NextSlotRespPiece) THEN
			M_ExeAction := E_ErrorIdCmd.ERRORID_InvalidExchangeOption;
			RETURN;
		END_IF
		
		IF fbObjectDirectory.M_ObjIsMzTool(refActionData.nObject) THEN //Object gültiges MzTool?
			pMzTool := fbObjectDirectory.M_GetObjPointer(refActionData.nObject);
		ELSE 
			M_ExeAction := E_ErrorIdCmd.ERRORID_UnsuitableObject;  //Error
			RETURN;
		END_IF
		
		CASE pMzTool^.P_eObjectType OF
			E_ObjectType.OBJECTTYPE_Luer:
				pLuer := pMzTool;
				rSumDockOffset := pLuer^.P_rDockOffset;
			E_ObjectType.OBJECTTYPE_TriplePip:
				pTriplePip := pMzTool;
				rSumDockOffset := pTriplePip^.P_rDockOffset;
			E_ObjectType.OBJECTTYPE_VacuumHandler:
				pVacuumHandler := pMzTool;
				rSumDockOffset := pVacuumHandler^.P_rDockOffset;			
			E_ObjectType.OBJECTTYPE_pHElectrode:
				ppHElectrode := pMzTool;
				//Dockoffset?
			E_ObjectType.OBJECTTYPE_StampSupport:
				pStampSupport := pMzTool;
			E_ObjectType.OBJECTTYPE_Gripper:
				pGripper := pMzTool;
		ELSE
			rSumDockOffset := 0;
		END_CASE
		
		pReactor := 0;
		pPowderStation :=0;
 
		IF fbObjectDirectory.M_ObjIsTarget(refActionData.nTarget) THEN //Target gültig?
			pTarget := fbObjectDirectory.M_GetObjPointer(refActionData.nTarget);
			//Slot ermitteln
			IF fbObjectDirectory.M_ObjIsRack(pTarget^.P_nObjectID) THEN //Target ein Rack?
				IF pTarget^.P_eObjectType = E_ObjectType.OBJECTTYPE_VialRackClosed THEN
					M_ExeAction := E_ErrorIdCmd.ERRORID_UnsuitableTarget;
					RETURN;
				END_IF
				pRack := pTarget;
				IF eExchangeOption = E_ExchangePieceOption.Slot THEN
					pPieceSlot := pRack^.M_GetSlot(DINT_TO_UINT(refActionData.aParams[1]));
					IF pPieceSlot = 0 THEN //Error
						M_ExeAction := E_ErrorIdCmd.ERRORID_InvalidTargetSlot;
						RETURN;
					END_IF
				ELSIF eExchangeOption = E_ExchangePieceOption.NextSlotRespPiece THEN
					IF bTakePiece THEN
						pPieceSlot := pRack^.M_GetNextFreshPieceSlot(pMzTool^.M_GetXYRange());
						IF pPieceSlot = 0 THEN //Error
							M_ExeAction := E_ErrorIdCmd.ERRORID_NoFreshPieceAvailable;
							RETURN;
						END_IF
					ELSE
						pPieceSlot := pRack^.M_GetNextFreeSlot(pMzTool^.M_GetXYRange());
						IF pPieceSlot = 0 THEN //Error
							M_ExeAction := E_ErrorIdCmd.ERRORID_NoFreeSlotAvailable;
							RETURN;
						END_IF
					END_IF
					//Überprüfen, ob Tool das Slot erreichen kann.
					//Wenn nicht, dann nächsten Slot holen.
					//Oder lieber den Bereich mit übergeben, in dem ein freier Slot verfügbar ist
					//Tools haben Props, welche die Min/Max-Pos zurückgeben
					
					refActionData.aParams[1] := pPieceSlot^.nNr;
				END_IF
			ELSIF pTarget^.P_eObjectType = E_ObjectType.OBJECTTYPE_Reactor THEN //Target ein Reaktor?
				pReactor := pTarget;
				IF eExchangeOption = E_ExchangePieceOption.Slot THEN
					pPieceSlot := pReactor^.M_GetSlot(DINT_TO_UINT(refActionData.aParams[1]));
					IF pPieceSlot = 0 THEN //Error
						M_ExeAction := E_ErrorIdCmd.ERRORID_InvalidTargetSlot;
						RETURN;
					END_IF					
				ELSIF eExchangeOption = E_ExchangePieceOption.NextSlotRespPiece THEN
					pPieceSlot := pReactor^.M_GetSlot(1);
				END_IF
			ELSIF pTarget^.P_eObjectType = E_ObjectType.OBJECTTYPE_PowderStation THEN //Target eine PowderStation?
				pPowderStation := pTarget;
				IF eExchangeOption = E_ExchangePieceOption.Slot THEN
					pPieceSlot := pPowderStation^.M_GetSlot(DINT_TO_UINT(refActionData.aParams[1]));
					IF pPieceSlot = 0 THEN //Error
						M_ExeAction := E_ErrorIdCmd.ERRORID_InvalidTargetSlot;
						RETURN;
					END_IF					
				ELSIF eExchangeOption = E_ExchangePieceOption.NextSlotRespPiece THEN
					pPieceSlot := pPowderStation^.M_GetSlot(1);
				END_IF				
			ELSIF pTarget^.P_eObjectType = E_ObjectType.OBJECTTYPE_SeptumWaste THEN //Target ein SeptumWaste?
				;
			END_IF
		ELSE
			M_ExeAction := E_ErrorIdCmd.ERRORID_UnsuitableTarget;  //Error
			RETURN;
		END_IF
		
		//Piece ermitteln
		pPiece := 0;
		IF bTakePiece THEN //Take, Piece wird vom Slot ermittelt
			IF pPieceSlot^.P_pPiece > 0 THEN
				pPiece := pPieceSlot^.P_pPiece^.P_pLatestChild;
			END_IF
		ELSE //Drop, Piece wird vom Tool ermittelt
			IF pMzTool^.P_pPiece > 0 THEN
				pPiece := pMzTool^.P_pPiece^.P_pLatestChild;
			END_IF
		END_IF
		
		IF pPiece = 0 THEN
			M_ExeAction := E_ErrorIdCmd.ERRORID_NoPieceDetermined;
			RETURN;
		END_IF
		
		rSumDockOffset := rSumDockOffset + pPiece^.P_rDockOffset;
		
		M_ExeAction := pMzTool^.M_CheckAction(refActionData, pPiece); //Action mit MzTool ausführbar?
		IF M_ExeAction > 0 THEN //Error
			RETURN;
		END_IF
		
		//Weitere Bedingungen des Targets checken		
		M_ExeAction := pTarget^.M_CheckAction(refActionData, pPiece); //Action mit Target ausführbar?
		IF M_ExeAction > 0 THEN
			RETURN;
		END_IF
		
		bExchangeNeedle := FALSE;
		bExchangeSeptum := FALSE;
		bExchangeTip := FALSE;
		bExchangeStamp := FALSE;
		bExchangeVial := FALSE;
		bExchangepHCap := FALSE;
		
		CASE pPiece^.P_eObjectType OF
			E_ObjectType.OBJECTTYPE_Needle:
				bExchangeNeedle := TRUE;
			E_ObjectType.OBJECTTYPE_Septum:
				bExchangeSeptum := TRUE;
			E_ObjectType.OBJECTTYPE_Tip:
				bExchangeTip := TRUE;
			E_ObjectType.OBJECTTYPE_Stamp:
				pStampMagazine := pTarget;
				bExchangeStamp := TRUE;
			E_ObjectType.OBJECTTYPE_Vial:
				bExchangeVial := TRUE;
			E_ObjectType.OBJECTTYPE_pHElectrodeCap:
				ppHElectrCapRack := pTarget;
				bExchangepHCap := TRUE;
		ELSE
			RETURN;
		END_CASE
 
	E_Action.ACTION_GetPipSample:
		IF fbObjectDirectory.M_ObjIsMzTool(refActionData.nObject) THEN //Object gültiges MzTool?
			pMzTool := fbObjectDirectory.M_GetObjPointer(refActionData.nObject);
		ELSE 
			M_ExeAction := E_ErrorIdCmd.ERRORID_UnsuitableObject;  //Error
			RETURN;
		END_IF
		
		IF fbObjectDirectory.M_ObjIsTarget(refActionData.nTarget) THEN //Target gültig?
			pTarget := fbObjectDirectory.M_GetObjPointer(refActionData.nTarget);
			IF pTarget^.P_eObjectType = E_ObjectType.OBJECTTYPE_Mtp THEN //derzeit nur mit Mtp ausführbar
				pMtp := pTarget;	
			ELSE
				M_ExeAction := E_ErrorIdCmd.ERRORID_UnsuitableTarget;  //Error
				RETURN;
			END_IF
		ELSE
			M_ExeAction := E_ErrorIdCmd.ERRORID_UnsuitableTarget;  //Error
			RETURN;
		END_IF
		
		M_ExeAction := pMzTool^.M_CheckAction(refActionData, pTarget); //Action mit MzTool ausführbar?
		IF M_ExeAction > 0 THEN
			RETURN;
		END_IF
		
		nCol := DINT_TO_UINT(refActionData.aParams[1]);
		nRow := DINT_TO_UINT(refActionData.aParams[2]);
		
		//pMzToolSpec := pMzTool;
		
		//Tool ein TwinPipHolder? -> FirstPip muss konfiguriert sein
		//-> SecondPip auch konfiguriert?
		IF pMzTool^.P_eObjectType = E_ObjectType.OBJECTTYPE_TwinPiezoHolder THEN
			//Mtp muss einen Wellabstand von 9mm haben 96er
			IF (pMtp^.P_rSpaceRows > 9500) OR (pMtp^.P_rSpaceRows < 8500) THEN
				M_ExeAction := E_ErrorIdCmd.ERRORID_MtpRowRiskOfCrash;
				RETURN;
			END_IF
			
			pTwinPiezoHolder := pMzTool;
			IF (pTwinPiezoHolder^.P_pPiezoPipFirst = 0) OR (pTwinPiezoHolder^.P_pPiezoPipSecond = 0) THEN
				M_ExeAction := E_ErrorIdCmd.ERRORID_NotAllPipettesConfigured;
				RETURN;
			ELSE
				//Checken, ob Zeile für Second gültig ist
				IF nRow < 3 THEN //SecondPip würde nicht mehr in Well treffen
					M_ExeAction := E_ErrorIdCmd.ERRORID_MtpRowRiskOfCrash;
					RETURN;
				END_IF
			END_IF
			//pMzTool := pTwinPiezoHolder^.P_pPiezoPipFirst;
		ELSIF pMzTool^.P_pParentMzTool^.P_eObjectType = E_ObjectType.OBJECTTYPE_TwinPiezoHolder THEN
			//Kann eintreten, wenn GetPipSample auf eine einzelne Pipette des TwinPipHolders ausgeführt wird
			//Crash der CoPipette mit Mtp verhindern
			pTwinPiezoHolder := pMzTool^.P_pParentMzTool;
			IF pMzTool = pTwinPiezoHolder^.P_pPiezoPipFirst THEN
				IF nRow < 3 THEN
					M_ExeAction := E_ErrorIdCmd.ERRORID_MtpRowRiskOfCrash;
					RETURN;
				END_IF
			ELSIF pMzTool = pTwinPiezoHolder^.P_pPiezoPipSecond THEN
				IF (nRow + 2) > pMtp^.P_nRows THEN
					M_ExeAction := E_ErrorIdCmd.ERRORID_MtpRowRiskOfCrash;
					RETURN;
				END_IF
			END_IF
		END_IF

		nQuantity1 := refActionData.aParams[3];
		nFlow1 := refActionData.aParams[4];
		nTime := DINT_TO_DWORD(refActionData.aParams[5]);
		nQuantity2 := refActionData.aParams[6];	//Quantity Airgap
		bGetPipSample_SwitchBypass := DINT_TO_BOOL(refActionData.aParams[7]);
		IF pMzTool^.P_eObjectType = E_ObjectType.OBJECTTYPE_PiezoPip OR pMzTool^.P_eObjectType = E_ObjectType.OBJECTTYPE_TwinPiezoHolder THEN
			bGetPipSample_ActivatePiezo := DINT_TO_BOOL(refActionData.aParams[8]);
		ELSE
			bGetPipSample_ActivatePiezo := FALSE;
		END_IF
		
		(*IF bGetPipSample_SwitchBypass THEN
			nQuantity2 := 0; //Quantity Airgap auf "0"
		END_IF*)
		
	E_Action.ACTION_InsertTool:
		IF fbObjectDirectory.M_ObjIsMzTool(refActionData.nObject) THEN //Gültiges MzTool?
			pMzTool := fbObjectDirectory.M_GetObjPointer(refActionData.nObject);
		ELSE 
			M_ExeAction := E_ErrorIdCmd.ERRORID_UnsuitableObject;  //Error
			RETURN;
		END_IF
		
		IF fbObjectDirectory.M_ObjIsTarget(refActionData.nTarget) THEN //Gültiges Target?
			pTarget := fbObjectDirectory.M_GetObjPointer(refActionData.nTarget);
		ELSE
			M_ExeAction := E_ErrorIdCmd.ERRORID_UnsuitableTarget;  //Error
			RETURN;
		END_IF
		
		M_ExeAction := pMzTool^.M_CheckAction(refActionData, pTarget); //Ausführbar mit MzTool?
		IF M_ExeAction > 0 THEN
			RETURN;
		END_IF
		
		M_ExeAction := pTarget^.M_CheckAction(refActionData, pMzTool); //Ausführbar mit Target?
		IF M_ExeAction > 0 THEN
			RETURN;
		END_IF
		
		M_ExeAction := pMzTool^.M_AskSiblingForAction(E_Action.ACTION_MoveToTarget);
		IF M_ExeAction > 0 THEN
			RETURN;
		END_IF
		
		
		eTargetRef := DINT_TO_USINT(refActionData.aParams[1]);
		nInsertLevel := DINT_TO_USINT(refActionData.aParams[4]);
		
		IF (pTarget^.P_eObjectGroup AND E_ObjectGroup.OBJECTGROUP_Rack) = E_ObjectGroup.OBJECTGROUP_Rack THEN
			pRack := pTarget;
			pPieceSlot := pRack^.M_GetSlot(DINT_TO_UINT(refActionData.aParams[2]));
		ELSIF pTarget^.P_eObjectType = E_ObjectType.OBJECTTYPE_Reactor THEN
			pReactor := pTarget;
			pPieceSlot := pReactor^.M_GetSlot(DINT_TO_UINT(refActionData.aParams[2]));
		ELSIF pTarget^.P_eObjectType = E_ObjectType.OBJECTTYPE_Mtp THEN
			pMtp := pTarget;
		END_IF
		
		IF eTargetRef = E_TargetRef.TARGETREF_Slot THEN
			IF pPieceSlot = 0 THEN
				M_ExeAction := E_ErrorIdCmd.ERRORID_InvalidTargetSlot;
				RETURN;
			ELSE
 				nTargetCol := UINT_TO_USINT(pPieceSlot^.nNr);
				nTargetRow := 0;
			END_IF
		ELSIF eTargetRef = E_TargetRef.TARGETREF_TwoDimArray THEN
			nTargetCol := DINT_TO_USINT(refActionData.aParams[2]);
			nTargetRow := DINT_TO_USINT(refActionData.aParams[3]);
		END_IF
	
	E_Action.ACTION_MeasureTool:
		bMeasureStamp := FALSE;
		bMeasureTarget := FALSE;
		bMeasureTip := FALSE;
		
		eMeasTipOption := DINT_TO_USINT(refActionData.aParams[2]);
		
		IF fbObjectDirectory.M_ObjIsTarget(refActionData.nTarget) THEN //Gültiges Target?
			pTarget := fbObjectDirectory.M_GetObjPointer(refActionData.nTarget);
		ELSE
			M_ExeAction := E_ErrorIdCmd.ERRORID_UnsuitableTarget;  //Error
			RETURN;
		END_IF		
	
		pMzTool := fbObjectDirectory.M_GetObjPointer(refActionData.nObject);
		IF pMzTool = 0 THEN
			M_ExeAction := E_ErrorIdCmd.ERRORID_ObjectNotExists;
			RETURN;
		END_IF
		
